(*============================================================================================*)		
(* Collision detection, soll verhinddern, dass nicht gesendet wird, wenn Daten im Empfangsüpuffer sind *)
(* Receive Collision Dectetion *)
bRXCollisionDetected :=	(I_pRxBuffer^.Count > INT_TO_UINT(iMaxBufferBlocking) 
						OR I_pRxBuffer^.FreeByte < (301 -INT_TO_UINT(iMaxBufferBlocking))
						OR I_pRxBuffer^.blocked
						OR I_pRxBuffer^.Error <> 0
						OR fbReceive.StringReceived
						(*OR sReceivedString <> ''*))
						AND bUseRXCollisionDetection;
						
(* Transmit Collision Detection *)
bTXCollisionDetected :=	(I_pTxBuffer^.Count > INT_TO_UINT(iMaxBufferBlocking) 
						OR I_pTxBuffer^.FreeByte < (301 -INT_TO_UINT(iMaxBufferBlocking))
						OR I_pTxBuffer^.blocked
						OR I_pTxBuffer^.Error <> 0)
						AND bUseTXCollisionDetection;
						
(* Collision Detection Verzögern *)						
tonCollisionFree(
	IN := 	NOT bRXCollisionDetected
			AND NOT bTXCollisionDetected,
	PT := 	tVerzCollisionDetect,
	Q =>	bCollisionFree);

(*============================================================================================*)	
(* Ping Intervall Timer *)		
tonPingIntervall(
	IN := I_bAutoPing
			AND NOT bPingStart,
	PT := I_tAutoPingTime);

tonPingVerz(
	PT := I_tVerzPing);	
	
(*============================================================================================*)	
(* Busbelastungstest *)	
bBusBelastungstest := I_bBusBelastungstest;
sReceivedMEMString:='';

(*============================================================================================*)	
(* Anzahl der gefüllten FiFo Zeilen *)
icntFiFo := 0;
iCntFiFoDone := 0;

FOR i := 1 TO cMaxRowCMDFiFo BY 1 DO 
	
	IF i <= I_nMaxDevices
	THEN
		IF (I_sSendCmdFiFo[i]<> '')
		THEN
			icntFiFo := icntFiFo +1;
		END_IF
	END_IF
	
	(* Zählen wie viele Dones gesetzt sind
		wenn alle True sind, ist komplett fertig gesendet *)
	IF i <= I_nMaxDevices
	THEN
		IF Q_bSendDoneFiFo[i]
		THEN
			iCntFiFoDone := iCntFiFoDone +1;
		END_IF
	END_IF
END_FOR

(* Alle FiFo Rows Done *)
bFiFoDone := iCntFiFoDone = I_nMaxDevices;
tonFiFoDoneTimeout.IN :=	NOT bFiFoDone
							AND iStepFiFo = 0;

(*============================================================================================*)	
(* Manuelles Senden *)
rTrigSendManuell(
	CLK := I_bSendManuell);

(*============================================================================================*)
CASE iStepFiFo OF
-1:	sStep := 'FiFo INIT';
	bFirstCycle := FALSE;
	Q_bBusy := FALSE;
	bPingStart := FALSE;
	iFiFoRow := 1;
	iPingRow := 1;
	
	FOR h := 1 TO cMaxRowCMDFiFo BY 1 DO
		IF h <= I_nMaxDevices
		THEN
			Q_bSendDoneFiFo[h] :=TRUE;
		END_IF
	END_FOR
	
	iStepFiFo := 0;

(*============================================================================================*)
0:	sStep := 'Warten, dass FiFo gefüllt wird';
		
	iFiFoRow := 1;
	
	IF iPingRow <= 0
	THEN
		iPingRow := 1;
	END_IF
	
	bStringSend := FALSE;
	Q_bBusy := FALSE;
	tonPingVerz.IN := FALSE;
		
	(* Wenn die Intervall Zeit abgelaufen ist Ping Start setzen *)
	IF tonPingIntervall.Q
	THEN
		bPingStart := TRUE;
	END_IF
	
	(* Notfallschaltung, falls mal ein bDone hängt
		zb. durch Gerätebaustein fehler *)
	IF tonFiFoDoneTimeout.Q
	THEN
		dwCntTimeout := dwCntTimeout+1;
		FOR h := 1 TO I_nMaxDevices BY 1 DO
			Q_bSendDoneFiFo[h] :=TRUE;
		END_FOR
	END_IF
					
	IF bFirstCycle
	THEN
		iStepFiFo := -1;
	ELSE
		IF bCollisionFree
		THEN
			IF icntFiFo > 0
				OR  bBusBelastungstest
				OR I_bManuellMode
			THEN
				(* Normaler Sendevorgang TX *)
				Q_bBusy := TRUE;
				iStepFiFo := 1;
			ELSE
				IF bPingStart
					OR iPingRow < I_nMaxDevices	(* Ping wurde unterbrochen *)
				THEN
					IF iPingRow < I_nMaxDevices
					THEN
						(* Fifo Zeile wieder auf die gespeicherte Ping zeile setzen, weil unterbrochen wurde *)
						iFiFoRow := iPingRow; 
					ELSE
						(* fifo Zeile 1 setzen, weil ende erreicht *)
						iFiFoRow := 1; 
					END_IF
					
					(* Globalen Merker Setzen, dass Ping aktiv ist *)
					bGlobalPingActive := TRUE;
					
					(* Ping senden TX*)
					iStepFiFo := 10;	
				END_IF
			END_IF
		END_IF
	END_IF
	
(*============================================================================================*)	
1:	sStep := 'Prüfen ob STRING in FiFo Zeile gefüllt*';
	
	IF I_bSearchMode
	THEN
		sStep :=fbRS485Search.Q_sState;
	END_IF
	
	(* Manueller Modus *)
	IF I_bManuellMode
	THEN
		(* Prüfen ob in der Zeile etwas steht *)
		IF I_sSendCmdManuell <>''
			AND rTrigSendManuell.Q
			AND NOT I_bSearchMode
		THEN
			IF bCollisionFree
			THEN
				(* Normaler Sendevorgang TX *)
				sString :=	I_sSendCmdManuell; 
				bStringSend := TRUE;
				Q_bDone := FALSE;
				Q_bError := FALSE;
				iStepFiFo := iStepFiFo+1;
			END_IF
		END_IF
		(* Prüfen ob in der Zeile etwas steht *)
		IF I_bSearchMode
			AND fbRS485Search.Q_bSend
		THEN
			IF bCollisionFree
			THEN
				(* Suchmode Sendevorgang TX *)
				sString :=	fbRS485Search.Q_sSearchString; 
				bStringSend := TRUE;
				Q_bDone := FALSE;
				Q_bError := FALSE;
				iStepFiFo := iStepFiFo+1;
			END_IF
		END_IF
	ELSE
		(* Prüfen ob in der ausgewählten Zeile etwas steht *)
		sStringSend :=	I_sSendCmdFiFo[iFiFoRow]; 
		IF I_sSendCmdFiFo[iFiFoRow] = ''
		THEN
			IF iFiFoRow< I_nMaxDevices
			THEN
				iFiFoRow := iFiFoRow+1; (* Nächste Zeile, bis etwas drin Steht *)
			ELSE
				IF bBusBelastungstest
				THEN
					sStringSend :=	CONCAT(F_ToCHR(I_sStartZeichen),'ServiceTOOL-BUSBELASTUNGSTEST-BURSTFIREMODE');
					sStringSend :=	CONCAT(sStringSend,F_ToCHR(I_sEndZeichen));
					(* Senden *)
					
					IF  bCollisionFree
					THEN
						(* Busbelastungstest Sendevorgang TX *)
						sStep := 'Prüfe ob Senden noch aktiv ist';
						bStringSend := TRUE;
						sString :=	sStringSend;
						Q_bDone := FALSE;
						Q_bError := FALSE;
						iStepFiFo := iStepFiFo+1;
					END_IF
				ELSE
					(* Alle Zeilen Abgearbeitet *)
					iStepFiFo := 0;	
				END_IF
			END_IF
		ELSE
		(* Senden *)
		Q_bSendDoneFiFo[iFiFoRow] :=FALSE;
		
			IF bCollisionFree
			THEN
				(* Normaler Sendevorgang TX *)
				sStep := 'Prüfe ob Senden noch aktiv ist';
				bStringSend := TRUE;
				sString :=	sStringSend;
				Q_bDone := FALSE;
				Q_bError := FALSE;
				iStepFiFo := iStepFiFo+1;
			END_IF
		END_IF
	END_IF
	
(*============================================================================================*)		
2:	sStep := 'Starte Senden';
	Q_bBusy := TRUE;
	tonTimeout.IN := fbSend.Busy;
	
	IF NOT fbSend.Busy
		AND NOT fbReceive.StringReceived
	THEN	
		(* Normaler Sendevorgang TX *)
		sString := '';
		tonSend.IN := FALSE;
		bStringSend := FALSE;
		iStepFiFo := iStepFiFo+1;
	ELSIF
		(fbSend.Error >0)
		AND NOT (fbSend.Error = 2)
	THEN
		sStep := CONCAT('ERROR-',sStep);
		sStep := CONCAT(sStep,'- ');
		sStep := CONCAT(sStep,INT_TO_STRING(fbSend.Error));
		iStepFiFo := -2;
	ELSIF
		tonTimeout.Q
	THEN
		sStep := CONCAT('ERROR- Timeout',sStep);
		iStepFiFo := -2;
	END_IF
	
(*============================================================================================*)		
3:	(* Senden*)		
	Q_bSendDoneFiFo[iFiFoRow] :=TRUE;
	
	IF iFiFoRow< I_nMaxDevices
		AND NOT I_bSearchMode
	THEN
		iFiFoRow := iFiFoRow+1;
		iStepFiFo := 1;
	ELSE
		Q_bDone := TRUE;
		
		IF (NOT fbRS485Search.Q_bSend
			AND I_bSearchMode)
			OR NOT I_bSearchMode
		THEN
			iStepFiFo := 0;
		END_IF
	END_IF
	
(*============================================================================================*)	
(* Ping Senden Ablauf *)
(*============================================================================================*)	
10:	sStep := 'Sende Ping*';
	
	tonPingVerz.IN := FALSE;
	
	(* Ping String erstellen *)
	sStringSend:=	CONCAT(F_ToCHR(I_sStartZeichen),DINT_TO_STRING(I_stDeviceIdent[iFiFoRow].diID));
	sStringSend :=	CONCAT(sStringSend,'.');
	sStringSend :=	CONCAT(sStringSend ,I_stDeviceIdent[iFiFoRow].sPingIdent); 
	sStringSend :=	CONCAT(sStringSend,F_ToCHR(I_sEndZeichen));
	
	IF I_stDeviceIdent[iFiFoRow].sPingIdent = ''
		OR I_stDeviceIdent[iFiFoRow].diID = 0
	THEN
		IF iFiFoRow < I_nMaxDevices
		THEN
			iFiFoRow := iFiFoRow+1; (* Nächste Zeile, bis etwas drin Steht *)
		ELSE
			bPingStart := FALSE;
			iPingRow := I_nMaxDevices;
			iStepFiFo := 0;	(* Alle Zeilen Abgearbeitet *)
		END_IF
	ELSE
	(* Senden *)	
		IF bCollisionFree
		THEN
			sStep := 'Prüfe ob Senden noch aktiv ist';
			bStringSend := TRUE;
			sString :=	sStringSend;
			Q_bDone := FALSE;
			Q_bError := FALSE;
			iStepFiFo := iStepFiFo+1;
		END_IF
	END_IF
	
(*============================================================================================*)		
11:	sStep := 'Starte Senden';
	Q_bBusy := TRUE;
	tonTimeout.IN := fbSend.Busy;
	
	IF NOT fbSend.Busy
		(*AND NOT fbReceive.StringReceived*)
	THEN
		tonSend.IN := FALSE;
		bStringSend := FALSE;
				
		IF NOT fbReceive.StringReceived
			AND bCollisionFree
		THEN
			iStepFiFo := iStepFiFo+1;
		END_IF
		
	ELSIF
		(fbSend.Error >0)
		AND NOT (fbSend.Error = 2)
	THEN
		sStep := CONCAT('ERROR-',sStep);
		sStep := CONCAT(sStep,'- ');
		sStep := CONCAT(sStep,INT_TO_STRING(fbSend.Error));
		iStepFiFo := -2;
	ELSIF
		tonTimeout.Q
	THEN
		sStep := CONCAT('ERROR- Timeout',sStep);
		iStepFiFo := -2;
	END_IF
	
(*============================================================================================*)		
12:	(* Senden*)		
	(* Nur speichern wenn auch wirklich eine ID vorhanden ist *)	
	IF I_stDeviceIdent[iFiFoRow].sPingIdent = ''
		OR I_stDeviceIdent[iFiFoRow].diID = 0
	THEN
		IF iFiFoRow < I_nMaxDevices
		THEN
			iFiFoRow := iFiFoRow+1; (* Nächste Zeile, bis etwas drin Steht *)
		ELSE
			bGlobalPingActive := FALSE;
			bPingStart := FALSE;
			iPingRow := I_nMaxDevices;
			iStepFiFo := 0;	(* Alle Zeilen Abgearbeitet *)
		END_IF
	ELSE
		IF iFiFoRow < I_nMaxDevices
		THEN
			iFiFoRow := iFiFoRow+1;
			iPingRow := iFiFoRow; (* Zeile speichern *)
			iStepFiFo := 13;	(* Falls das warten Deaktiviert werden soll, kann hier einfach in 10 gesprungen werden *)
		ELSE
			bPingStart := FALSE; (* Letzte Ping Zeile erreicht, Timer zurücksetzen  *)
			iPingRow := I_nMaxDevices;
			iStepFiFo := 13;
		END_IF
	END_IF
(*============================================================================================*)		
13:	(* Optionale Wartezeit zwischen jedem Ping*)		
	tonPingVerz.IN := TRUE;
			
	IF tonPingVerz.Q
	THEN
		IF NOT fbReceive.StringReceived
			AND bCollisionFree
		THEN
			tonPingVerz.IN := FALSE;
			
			IF iFiFoRow < I_nMaxDevices
			THEN
				iStepFiFo := 10; (* nächsten Ping senden *)
			ELSE
				bGlobalPingActive := FALSE;
				iStepFiFo := 0;
			END_IF
		END_IF
	ELSE
		(* Prüfen ob ein Sendeauftrag anliegt *)
		IF icntFiFo >0
		THEN
			tonPingVerz.IN := FALSE;
			iStepFiFo := 0; (* Sende FiFo leeren *)
		END_IF  
	END_IF
ELSE
(*============================================================================================*)
	Q_bError := TRUE;
	Q_bBusy := FALSE;
	bBusyMem := FALSE;
	tonTimeout.IN := FALSE;
	
	IF I_bReset
	THEN
		iStepFiFo := 0;
	END_IF
END_CASE

(*============================================================================================*)	
(* Nur Senden, wenn nicht Empfangen wird *)
IF bStringSend
THEN
	IF bActivateSend
	THEN
		(* Senden *)
		fbSend(
			SendString:= 	sString,
			TXbuffer:= 		I_pTxBuffer^);
	END_IF
	
ELSE
	IF bActivateReceive
	THEN
		(* Empfangen *)
		ac00_Receive();
	END_IF
END_IF

(*============================================================================================*)	
(* Empfangsmerker 0 Setzen am ende Eines Zyklus *)
Q_sReceiveString := sReceivedMEMString;

(*============================================================================================*)	
(* Busauslastung tracken*)
ac99_Diagnose();

(*============================================================================================*)	
(* StatusStruktur für Visu *)
Q_sState :=	sStep;
Q_stStates.bBusy				:=	Q_bBusy;
Q_stStates.bDone				:=	Q_bDone;
Q_stStates.bError				:=	Q_bError;
Q_stStates.iFiFoCount			:=	icntFiFo;
Q_stStates.iFiFoRow				:=	iFiFoRow;
Q_stStates.lrBusAuslastung		:=	Q_lrBusAuslastung;
Q_stStates.sReceiveString 		:=	Q_sReceiveString;
Q_stStates.sSendString 			:=	sString;
Q_stStates.sState 				:=	Q_sState;

(*============================================================================================*)	
(* RS485 Telegramm Logging *)
fbRS485Logger(
	I_bExecute:= 		I_bLogger,						(* oder eine externe Variable *)
	I_bReset:=			I_bResetLog,	
	I_sTxTelegram:= 	sString,
	I_sRxTelegram:= 	sReceivedMEMString);

ACTION ac00_Receive:
(*============================================================================================*)	
(* Empfangen *)

CASE iStepReceive OF		
0:	fbReceive(
		Prefix := 			F_ToCHR(I_sStartZeichen),
		Suffix := 			F_ToCHR(I_sEndZeichen),
		Timeout:= , 
		Reset:= , 
		StringReceived=> , 
		Busy=> , 
		Error=> , 
		RxTimeout=> , 
		ReceivedString:= 	sReceivedString, 
		RXbuffer:= 			I_pRxBuffer^);
		
	IF fbReceive.StringReceived
	THEN
		iStepReceive := 1;
		sReceivedMEMString := sReceivedString;
	END_IF
	
1:	sReceivedString := '';
	iStepReceive := 0;

	
END_CASE
END_ACTION

ACTION ac99_Diagnose:
(*============================================================================================*)	
(* Busauslastung Prüfen *)

fbBusAuslastung(
	I_bExcecute:= 	bBusAuslastung, 
	I_nWert:= 		UINT_TO_LREAL(I_pTxBuffer^.Count), 
	I_nFilterWert:= 50, 
	Q_nFilter=> 	Q_lrBusAuslastung);
	
	
fbRS485Search(
	I_bStartSearch:= 	I_bSearchMode, 
	I_diStartID:= , 
	I_diMaxID:= , 
	I_sStartZeichen:= 	I_sStartZeichen, 
	I_sEndZeichen:= 	I_sEndZeichen, 
	I_tWait:= , 
	I_StringReceived:= 	sReceivedMEMString, 
	Q_bSend=> , 
	Q_sSearchString=> );
END_ACTION

END_FUNCTION_BLOCK

// ---- POUs/RS485_Hausbus_FB/00_RS485 COM/RS485_Master/fb_RS485Logger.TcPOU
(*======================================================================================================================================*)
(*//=============================================================================\\
||  _   _ _  __  _         _                        _   _                      ||
|| | \ | | |/ / / \  _   _| |_ ___  _ __ ___   __ _| |_(_) ___  _ __         ||
|| |  \| | ' / / _ \| | | | __/ _ \| '_ ` _ \ / _` | __| |/ _ \| '_ \        ||
|| | |\  | .  \/ ___ \ |_| | || (_) | | | | | | (_| | |_| | (_) | | | |       ||
|| |_| \_|_|\_\_/  \_\__,_|\__\___/|_| |_| |_|\__,_|\__|_|\___/|_| |_|       ||
||                                                                             ||
\\=============================================================================//*)
(*fb_RS485Logger: 	Einfaches Logging von RX und TX Telegrammen*)
(*
Date          	| Version    	| created under        	| Author          	| Remark *)
(*====================================================================================================================================================*)
(*11/01/2026   	| 1.00      		| TC3		  		| N. Kersting       | first release *)
(*11/01/2026   	| 1.01      		| TC3		  		| N.  Kersting       | Ringbuffer implementiert - neueste oben *)
(*11/01/2026   	| 1.02      		| TC3		  		| N.  Kersting       | Array wird geleert wenn Execute FALSE ist *)
(*12/01/2026   	| 1.03      		| TC3		  		| N.  Kersting       | Reset eingang zum zurücksetzen des gesamten Arrays *)
(*====================================================================================================================================================*)
FUNCTION_BLOCK fb_RS485Logger
VAR_INPUT
	I_bExecute				: BOOL := TRUE;								(* Enable/Disable Logging *)
	I_bReset				: BOOL;										(* Reset Log Buffer *)
	I_sTxTelegram			:STRING(255);								(* TX Telegramm zum Logging *)
	I_sRxTelegram			:STRING(255);								(* RX Telegramm zum Logging *)
END_VAR
VAR_OUTPUT
	Q_asLogBuffer			:ARRAY[1..50] OF STRING(255);				(* Log Buffer mit max.  200 Zeilen *)
	Q_iLogIndex				:INT;										(* Aktuelle Index Position *)
	Q_iLogCount				:INT;										(* Anzahl der geloggten Einträge *)
END_VAR
VAR
	sTxLast					: STRING(255) := '';						(* Letzter TX String zum Vergleich *)
	sRxLast					: STRING(255) := '';						(* Letzter RX String zum Vergleich *)
	bExecuteLast			: BOOL := TRUE;								(* Letzter Execute Status *)
	iWriteIndex				: INT := 1;									(* Schreibposition Ringbuffer *)
	iLogCount				:INT := 0;									(* Gesamtanzahl Logs *)
	sLogEntry				: STRING(255);								(* Temporärer Log Eintrag *)
	i, h					: INT;										(* Zähler *)

END_VAR

(*============================================================================================*)
(* Reset Log Buffer - leert das komplette Array *)
IF I_bReset
THEN
	FOR i := 1 TO 50 BY 1 DO
		Q_asLogBuffer[i] := '';
	END_FOR
	iLogCount := 0;
	sTxLast := '';
	sRxLast := '';
	RETURN;
END_IF

(*============================================================================================*)
(* Logging deaktiviert - nur schreiben pausieren *)
IF NOT I_bExecute
THEN
	RETURN;
END_IF

(*============================================================================================*)
(* TX Telegramm Logging *)
IF I_sTxTelegram <> '' 
	AND I_sTxTelegram <> sTxLast
THEN
	(* Alle Zeilen nach unten verschieben - rückwärts von 199 bis 1 *)
	FOR h := 49 TO 1 BY -1 DO
		Q_asLogBuffer[h + 1] := Q_asLogBuffer[h];
	END_FOR
	
	(* Neuer Eintrag oben *)
	sLogEntry := CONCAT('TX: ', I_sTxTelegram);
	Q_asLogBuffer[1] := sLogEntry;
	sTxLast := I_sTxTelegram;
	
	(* Counter erhöhen, aber max. 200 *)
	IF iLogCount < 50
	THEN
		iLogCount := iLogCount + 1;
	END_IF
END_IF

(*============================================================================================*)
(* RX Telegramm Logging *)
IF I_sRxTelegram <> '' 
	AND I_sRxTelegram <> sRxLast
THEN
	(* Alle Zeilen nach unten verschieben - rückwärts von 199 bis 1 *)
	FOR h := 49 TO 1 BY -1 DO
		Q_asLogBuffer[h + 1] := Q_asLogBuffer[h];
	END_FOR
	
	(* Neuer Eintrag oben *)
	sLogEntry := CONCAT('RX: ', I_sRxTelegram);
	Q_asLogBuffer[1] := sLogEntry;
	sRxLast := I_sRxTelegram;
	
	(* Counter erhöhen, aber max. 200 *)
	IF iLogCount < 50
	THEN
		iLogCount := iLogCount + 1;
	END_IF
END_IF

(*============================================================================================*)
(* Output Parameter aktualisieren *)
Q_iLogCount := iLogCount;

END_FUNCTION_BLOCK

// ---- POUs/RS485_Hausbus_FB/00_RS485 COM/RS485_Master/fb_RS485Startup.TcPOU
(*======================================================================================================================================*)
(*//=============================================================================\\
||  _   _ _  __  _         _                        _   _                      ||
|| | \ | | |/ / / \  _   _| |_ ___  _ __ ___   __ _| |_(_) ___  _ __         ||
|| |  \| | ' / / _ \| | | | __/ _ \| '_ ` _ \ / _` | __| |/ _ \| '_ \        ||
|| | |\  | . \/ ___ \ |_| | || (_) | | | | | | (_| | |_| | (_) | | | |       ||
|| |_| \_|_|\_\_/  \_\__,_|\__\___/|_| |_| |_|\__,_|\__|_|\___/|_| |_|       ||
||                                                                             ||
\\=============================================================================//
fb_RS485Startup:	Einfacher Baustein um die Hardware für die RS485 Haus-Bus vorzubereiten*)
(*
Date          	| Version    	| created under        	| Author          	| Remark *)
(*====================================================================================================================================================*)
(*13/05/2025   	| 1.00      		| TC3		  		| N.Kersting       | first release *)
(*18/08/2025   	| 1.01      		| TC3		  		| N.Kersting       | Startup über bExecute nun erneut Anwählbar*)
(*13/10/2025   	| 1.02      		| TC3		  		| N.Kersting       | Automatische Quittierung bei Busfehler*)
(*15/10/2025   	| 1.03      		| TC3		  		| N.Kersting       | Spannungsversorgung nun steuerbar über diesen Baustein*)
(*19/10/2025   	| 1.04      		| TC3		  		| N.Kersting       | Bugfix automatische Quittierung nach Busfehler nur bei Spannung Ok*)
(*====================================================================================================================================================*)
FUNCTION_BLOCK fb_RS485Startup
VAR_INPUT
	I_bExecute						:BOOL;
	I_bBusOK						:BOOL;
	I_bSpannungOk					:BOOL;
	I_bStandby						:BOOL;
	I_tStartupVerz					:TIME := T#2S;	(* Startup verzögert ausführen *)
END_VAR
VAR_IN_OUT
	IQ_InData	 					:KL6inData22B;
    IQ_OutData						:KL6outData22B;
END_VAR
VAR_OUTPUT
	Q_sState						:STRING;
	Q_bStartupDone					:BOOL;
	Q_bError						:BOOL;
	Q_bSpannungEin					:BOOL;
	Q_bSpannungAus					:BOOL;
	Q_stStates						:ST_RS485Startup_State;
END_VAR
VAR
	udBaudrate						:UDINT := 57600;
	byDataBits						:BYTE := 8;
	byStopBits						:BYTE := 1;
	
	tonStartupVerz					:ton;
	tonTimeout						:ton;
	fbSerialComReset				:ComReset;
	fComBufferReset					:ClearComBuffer;
	fbSerialConfig 					:KL6Configuration;  // Terminal-Konfiguration (Baud, Parität etc.)
	iStepStartup					:INT;
	rTrigStartupStart				:r_trig;
	bBusFehlerMerker				:BOOL;
END_VAR

tonStartupVerz(
	PT :=	I_tStartupVerz);

tonTimeout();	

rTrigStartupStart(CLK :=Q_bStartupDone
						AND I_bExecute
						AND I_bBusOK);
	
CASE iStepStartup OF 
(*=========================================================================*)
0:	tonTimeout.IN := FALSE;
	Q_bSpannungEin := FALSE;
	Q_bSpannungAus := FALSE;
	
	IF NOT Q_bError
		AND I_bBusOK
	THEN
		Q_sState := 'INIT';
	ELSIF
		NOT I_bBusOK
	THEN
		bBusFehlerMerker := TRUE;
		Q_bError := TRUE;
		Q_sState := 'Busverbindung nicht Ok';
	END_IF
	
	tonStartupVerz.IN := FALSE;
	
	fbSerialComReset(
		Execute:= 		FALSE);
		
	fbSerialConfig(
		Execute:= 		FALSE);
		
	(* Automatische Quittierung nach Busfehler *)
	IF bBusFehlerMerker
		AND I_bBusOK
		AND I_bSpannungOk
	THEN
		Q_bStartupDone := FALSE;
		iStepStartup := iStepStartup+1;
	END_IF
	
	IF I_bExecute
		AND I_bBusOK
		AND I_bSpannungOk
	THEN
		Q_bStartupDone := FALSE;
		iStepStartup := iStepStartup+1;
	ELSIF
		I_bExecute
		AND I_bBusOK
		AND NOT I_bSpannungOk
	THEN
		Q_bStartupDone := FALSE;
		iStepStartup := 100;
	END_IF

(*=========================================================================*)
1:	Q_sState := 'Warten auf Verzögerung';
	tonStartupVerz.IN := TRUE; 
	
	IF tonStartupVerz.Q
	THEN
		iStepStartup := iStepStartup+1;
	END_IF
	
(*=========================================================================*)
2:	Q_sState := 'Serielle Klemme Konfigurieren mit Haus-Bus Vorgaben';	
	
	fbSerialConfig(
		Execute:= 		TRUE, 
		Mode:= 			ComSerialLineMode_t.SERIALLINEMODE_KL6_22B_STANDARD,		 
		Baudrate:= 		udBaudrate, 
		NoDatabits:= 	byDataBits, 
		Parity:= 		ComParity_t.PARITY_EVEN,	 
		Stopbits:= 		byStopBits, 
		Handshake:= 	RS485_HALFDUPLEX, 
		ContinousMode:= , 
		pComIn := 		ADR(IQ_InData), 
		pComOut := 		ADR(IQ_OutData), 
		SizeComIn := 	SIZEOF(IQ_InData),
		Done=> , 
		Busy=> , 
		Error=> , 
		ErrorId=> );
	
	IF fbSerialConfig.Done
	THEN
		fbSerialConfig(
			Execute:= 		FALSE); 
			
		iStepStartup := 3;
	ELSIF
		fbSerialConfig.Error
	THEN
		Q_sState := 'Error fbSerialConfig ID: ';
		Q_sState := CONCAT(Q_sState,INT_TO_STRING(fbSerialConfig.ErrorID));
		iStepStartup := -2;	//Error
	END_IF

(*=========================================================================*)
3:	Q_sState := 'Serielle Klemme Reset Auführen';	
		
	fbSerialComReset(
		Execute:= 		TRUE, 
		pComIn := 		ADR(IQ_InData), 
		pComOut := 		ADR(IQ_OutData), 
		SizeComIn := 	SIZEOF(IQ_InData),
		Done=> , 
		Busy=> , 
		Error=> , 
		ErrorID=> );	
		
	IF fbSerialComReset.Done
	THEN
		iStepStartup := 999;
	ELSIF
		fbSerialComReset.Error
	THEN
		Q_sState := 'Error fbSerialComReset ID: ';
		Q_sState := CONCAT(Q_sState,INT_TO_STRING(fbSerialComReset.ErrorID));
		iStepStartup := -3;	//Error
	END_IF

(*=========================================================================*)
100:Q_sState := 'Spannung einschalten';
	tonTimeout.IN := TRUE;
	tonTimeout.PT := T#5S;
	
	Q_bSpannungEin := TRUE;

	IF 	I_bSpannungOk
	THEN
		Q_bSpannungEin := FALSE;
		tonTimeout.IN := FALSE;
		iStepStartup := 1;
	ELSIF
		tonTimeout.Q
	THEN
		Q_bSpannungEin := FALSE;
		tonTimeout.IN := FALSE;
		Q_sState := 'Timeout Spannung einschalten';
		iStepStartup := -100;
	END_IF

(*=========================================================================*)
200:Q_sState := 'Spannung ausschalten';
	tonTimeout.IN := TRUE;
	tonTimeout.PT := T#5S;
	
	Q_bSpannungAus := TRUE;

	IF 	NOT I_bSpannungOk
	THEN
		Q_sState := 'HausBus Spannung über Standby Ausgeschaltet. Startup Ausführen zum einschalten!';
		Q_bSpannungAus := FALSE;
		tonTimeout.IN := FALSE;
		iStepStartup := -201;	(* Standby *)
	ELSIF
		tonTimeout.Q
	THEN
		Q_bSpannungAus := FALSE;
		tonTimeout.IN := FALSE;
		Q_sState := 'Timeout Spannung ausschalten';
		iStepStartup := -200;
	END_IF
	
(*=========================================================================*)
999:Q_sState := 'Startup Ausgeführt!';	
	Q_bStartupDone := TRUE;
	Q_bError := FALSE;
	bBusFehlerMerker := FALSE;
	tonTimeout.IN := FALSE;
	Q_bSpannungEin := FALSE;
	Q_bSpannungAus := FALSE;
	
	IF NOT I_bBusOK
		OR NOT I_bSpannungOk
	THEN
		bBusFehlerMerker := TRUE;
		Q_bStartupDone := FALSE;
		iStepStartup := 0;
	END_IF
	
	IF I_bSpannungOk
		AND I_bStandby
	THEN
		Q_bStartupDone := FALSE;
		iStepStartup := 200;
	END_IF
	
	IF rTrigStartupStart.Q
	THEN
		Q_bStartupDone := FALSE;
		iStepStartup := 1;
	END_IF

ELSE
	(* ERROR *)
	Q_bError := TRUE;
	iStepStartup := 0;
END_CASE

(* StatusStruktur für Visu *)
Q_stStates.bBusOk				:=	I_bBusOK;
Q_stStates.bStartupDone			:=	Q_bStartupDone;
Q_stStates.bStartupError		:=	Q_bError;
Q_stStates.sStartupState		:=	Q_sState;

END_FUNCTION_BLOCK

// ---- POUs/RS485_Hausbus_FB/01_BusTaster/fb_TasterBus6F.TcPOU
(*======================================================================================================================================*)
(*//=============================================================================\\
||  _   _ _  __  _         _                        _   _                      ||
|| | \ | | |/ / / \  _   _| |_ ___  _ __ ___   __ _| |_(_) ___  _ __         ||
|| |  \| | ' / / _ \| | | | __/ _ \| '_ ` _ \ / _` | __| |/ _ \| '_ \        ||
|| | |\  | . \/ ___ \ |_| | || (_) | | | | | | (_| | |_| | (_) | | | |       ||
|| |_| \_|_|\_\_/  \_\__,_|\__\___/|_| |_| |_|\__,_|\__|_|\___/|_| |_|       ||
||                                                                             ||
\\=============================================================================//
fb_TasterBus6F:	Einfache RS485 Kommunikation für Haus-bus.de Komponenten zum testen 	
				Achtung: Bei dem 6 Fach Taster ist zu Beachten, dass es nur 4 Externe EA/s gibt also 4 LEDs und 4 Taster *)
(*
Date          	| Version    	| created under        	| Author          	| Remark *)
(*====================================================================================================================================================*)
(*29/04/2025   	| 1.00      		| TC3		  		| N.Kersting       | first release *)
(*02/05/2025   	| 1.01      		| TC3		  		| N.Kersting       | Events für die Buttons werden erfolgreich verarbeitet *)
(*02/05/2025   	| 1.02      		| TC3		  		| N.Kersting       | Events für Temp, Helligkeit, Fuehctigkeit erfolgreich Implementier *)
(*02/05/2025   	| 1.03      		| TC3		  		| N.Kersting       | Set Schrittkette für Reset und LED Helligkeit erfolgreich Implementier*)
(*02/05/2025   	| 1.04      		| TC3		  		| N.Kersting       | In und Out Strukturen Implementiert und Startup nach Reset *)
(*02/05/2025   	| 1.05      		| TC3		  		| N.Kersting       | Pingabgfrage*)
(*02/05/2025   	| 1.06      		| TC3		  		| N.Kersting       | Reset Startup Implementiert*)
(*03/05/2025   	| 1.07      		| TC3		  		| N.Kersting       | Ping wird nun bei PLC Reset auch gestaret und Execute wird richtig verwendet*)
(*04/05/2025   	| 1.08      		| TC3		  		| N.Kersting       | Hintergrundbeleuchtung und Zähler für die Tatser Implementiert *)
(*04/05/2025   	| 1.09      		| TC3		  		| N.Kersting       | Neuen Baustein zum Einheitlichen versenden von Telegrammen Implementiert *)
(*05/05/2025   	| 2.00      		| TC3		  		| N.Kersting       | Komplett neuen Baustein, mit Externer Receive Auswertung und neuem Ping Baustein *)
(*06/05/2025   	| 2.01      		| TC3		  		| N.Kersting       | Externe LEDs Implementiert *)
(*07/05/2025   	| 2.02      		| TC3		  		| N.Kersting       | Im Startup wird nun auf die Device ID geachtet *)
(*08/05/2025   	| 2.03      		| TC3		  		| N.Kersting       | Externe LEDs sind nun Umschaltbar/ LEDs oder normaler Ausgang (Betriefft die Hintergrundbeleuchtung) -> Weniger Busauslastung *)
(*09/05/2025   	| 2.04      		| TC3		  		| N.Kersting       | Ping Versuche Implementiert mit Globalen Parametern *)
(*09/05/2025   	| 2.05      		| TC3		  		| N.Kersting       | Ping für Taster nun Auch automatisch durch Empfang von sämtlichen Telegrammen*)
(*09/05/2025   	| 2.06      		| TC3		  		| N.Kersting       | Bugfix im Startup Angepasst! nur noch Hintergrundbeleuchtung setzen! *)
(*10/05/2025   	| 3.00      		| TC3		  		| N.Kersting       | Umstellung auf Externe FiFo Sendebaustein *)
(*13/05/2025   	| 3.01      		| TC3		  		| N.Kersting       | Viele Bugs gefixt, bei Änderung der Ausgängen wird nun eine Anforderung gesetzt  *)
(*13/05/2025   	| 3.02      		| TC3		  		| N.Kersting       | Test für Github *)
(*23/05/2025   	| 3.03      		| TC3		  		| N.Kersting       | Auto - Input Fault Detection implementiert (Wenn Taster zu lange aktiviert bleibt ) *)
(*28/05/2025   	| 3.04      		| TC3		  		| N.Kersting       | Neuen Einfachen Ping Baustein, welcher nicht sendet, nur auswertet implementiert *)
(*14/08/2025   	| 3.05      		| TC3		  		| N.Kersting       | Neuen Taster Eventbaustein, welcher deutlich weniger CPU Last verursacht  *)
(*27/08/2025   	| 4.00      		| TC3		  		| N.Kersting       | Neue Startupschrittkette sollte alle Eventbausteine auch Resetten  *)
(*28/08/2025   	| 5.00      		| TC3		  		| N.Kersting       | Komplett neue Evolutionsstufe, alle Hausbusgeräte werden nun vom fb_UniHBComOperator gesteuert  *)
(*28/08/2025   	| 5.01      		| TC3		  		| N.Kersting       | Etrster Test erfogreich *)
(*31/08/2025   	| 5.02      		| TC3		  		| N.Kersting       | Bugfix OP Mode wird angezeigt bei Init *)
(*03/09/2025   	| 5.03      		| TC3		  		| N.Kersting       | Events geben nun einen Zeitstempel und die differenz vom letzten Update aus *)
(*05/09/2025   	| 5.04      		| TC3		  		| N.Kersting       | Changecounter gibt nun die Anzahl der  Startups wieder *)
(*09/09/2025   	| 5.05      		| TC3		  		| N.Kersting       | Events aus der For-schleife geholt *)
(*29/09/2025   	| 5.06      		| TC3		  		| N.Kersting       | Inputfault detection für Ext eingänge deaktiviert für Bewegungsmelder *)
(*22/01/2026   	| 7.00      		| TC3		  		| N.Kersting       | Komplett überarbeitet mit umstellung auf Stringbuilder *)
(*25/01/2026   	| 7.01      		| TC3		  		| N.Kersting       | Eventbausteine alle komplett überarbeitet mit den neuen ASCII_RS485 Funktionen *)
(*08/06/2026   	| 8.00      		| TC3		  		| N.Kersting       | Vorbereitung für Bibliotheksfähigkeit, keine externen Referenzen mehr *)
(*20/09/2026   	| 9.00      		| TC3		  		| N.Kersting       | Selbsttest für Abfrage der eingänge *)
(*20/09/2026   	| 9.01      		| TC3		  		| N.Kersting       | Selbsttest Bugfix Schrittkette *)
(*20/09/2026   	| 9.02      		| TC3		  		| N.Kersting       | Selbsttest Bugfix Schrittkette *)
(*20/09/2026   	| 9.03      		| TC3		  		| N.Kersting       | Selfcheck nun nur, wenn Globaler Pingmerker nicht aktiv *)
(*20/09/2026   	| 9.04      		| TC3		  		| N.Kersting       | Kleine anpassung Autoping *)
(*====================================================================================================================================================*)
FUNCTION_BLOCK fb_TasterBus6F
VAR_INPUT
	I_bUsePing			:BOOL;
	I_tPingTime			:TIME := T#15S;
	I_tSelfCheckTime	:TIME := T#15S;
	
	I_bFiFoDone			:BOOL;
	I_FifoID			:INT;
	I_bPingStart		:BOOL;						(* Ping Done vom Vorheriegen*)
	I_bSelfCheck		:BOOL := FALSE;				(* 1x Eingänge prüfen Achtung Flanke!*)
	I_bSelfCheckAuto	:BOOL := FALSE;				(* Eingänge Automatisch Intervallsmäßig prüfen *)
	
	I_stInput			:ST_BusTaster6F_Input;
	I_StringReceived	:STRING(255);
END_VAR
VAR_OUTPUT
	Q_sFiFoSend			:STRING(255);
   	Q_stOutput			:ST_BusTaster6F_Output;
	Q_stCnt				:ST_BusTaster6F_Cnt;
END_VAR
VAR
(*----------------------------------------------*)
(* Interne Parameter*)
(*----------------------------------------------*)		
	bSetExecute			:BOOL := TRUE;				(* Aktiviert die Schrittketten, welche Telegramme versenden *)
	bCheckPing			:BOOL := TRUE;				(* Ping Checken Schrittkette Aktivieren *)
	bInputFaultDetect	:BOOL := TRUE;				(* Prüft die Eingänge ob sie zu lange geschaltet wurden und führt ein reset des eingangs aus *)
	
	sStartZeichen		:BYTE := 16#FD;				(* Startzeichen Präfix *)
	sEndZeichen			:BYTE := 16#FE;				(* Endzeichen Suffix *)
	
	tPingTimer			:TIME:= T#5S;				(* Zeit, bis wiederholend der Ping versendet wird *)
	tStartupLEDOn		:TIME:= T#4S;				(* Zeit, wie Lange die LEDS beim Startup kurz eingeschaltet werden *)
	tResetTimeout		:TIME:= T#10S;				(* Zeit, bis bei einem Reset es zu einem Fehler kommt, wenn kein Ping empfangen wird *)
	tResetReboot		:TIME:= T#10S;				(* Zeit, die nach einem Reset Abgewaretet wird damit das Gerät neustarten kann*)
	tStartupAfterReset	:TIME := T#5S;				(* Zeit, wann das Startup Zurückgesetzt wird, wenn der Ping verloren wird *)
	tInputFaultDetect	:TIME := T#10S;				(* Prüft die Eingänge ob sie zu lange geschaltet wurden und führt ein reset des eingangs aus *)
	
	tSelfCheckStatus	:TIME := T#15S;				(* Prüft die Externen u. Internen Eingänge zyklisch in diesem rythmus ab *)
(*----------------------------------------------*)
(* Strings *)
(*----------------------------------------------*)			
	sSendString			:STRING(255);
	sFiFoSend			:STRING(255);
	sReceived			:STRING(255);
	sLastSendString		:STRING(255);
	sStateReset			:STRING;
(*----------------------------------------------*)
(* Funktionsbausteine *)
(*----------------------------------------------*)
	fbUniHBComOperator	:fb_UniHBComOperator;
	fbBusTasterEventExt	:fb_BusTasterAdvancedEvent_6F;
	fbBusTasterEvent	:fb_BusTasterAdvancedEvent_6F;
	fbBusTempEvent		:fb_BusTempEvent;
	fbBusBrsEvent		:fb_BusBrsEvent;
	fbBusRhdEvent		:fb_BusRhdEvent;
	fbBusPingEvent		:fb_BusPingEvent;
(*----------------------------------------------*)
(* Indexe *)
(*----------------------------------------------*)	
	iStepSet			:INT;
	i,h,j,l,e			:INT;
	
	iDimmMem			:ARRAY[1..6] OF INT;
	iDimmMemExt			:ARRAY[1..6] OF INT;
	iDimmBGAnf			:INT;
	iDimmAnf			:ARRAY[1..6] OF INT;
	iDimmAnfExt			:ARRAY[1..6] OF INT;
	
	iDimmBgMem			:INT;
	cntChangesDimm		:INT;
	cntChangesDimmExt	:INT;
(*----------------------------------------------*)
(* Timer/Trigger *)
(*----------------------------------------------*)		
	r_TrigReset				:r_trig;		
	r_TrigCountBtn			:ARRAY[1..6] OF r_trig;
	
	tonResetTimeout			:ton;
	tonStepStartup			:ton;
	tonSelfCheck			:ton;
(*----------------------------------------------*)
(* Status *)
(*----------------------------------------------*)			
	bMemExt					:BOOL;
	bSendeAnforderung		:BOOL;
	bSendeAnforderungExt	:BOOL;
	bSendeAnforderungBG		:BOOL;
	bErrorReset				:BOOL;
	bResetBusy				:BOOL;
	bResetDone				:BOOL;
	bStartupDone			:BOOL;
	bEventStartupDone		:BOOL;
	bSelfCheckAnforderung	:BOOL;
	
	fbRS485HBStringBuilder	:fb_RS485HB_StringBuilder;
END_VAR

(*///////////////////////////////////////////////////////////*)
(* Parameter *)
tPingTimer :=			I_tPingTime;
bCheckPing :=			I_bUsePing;

(*///////////////////////////////////////////////////////////*)
(* Reset *)
r_TrigReset(CLK := 	I_stInput.bReset);

(*///////////////////////////////////////////////////////////*)
(* Ident beschreiben *)
fbUniHBComOperator.I_stIdent.bUseExtInputs 	:=	I_stInput.bExtInputs;
fbUniHBComOperator.I_stIdent.diID 			:=	I_stInput.diID;
fbUniHBComOperator.I_stIdent.sName 			:=	I_stInput.sName;

(*///////////////////////////////////////////////////////////*)
(*	Operator *)
fbUniHBComOperator(
	I_bExtInputs:= 			I_stInput.bExtInputs, 
	I_bExecute:= 			I_stInput.bExecute
							AND NOT r_TrigReset.Q, 
	I_bPing:= 				fbBusPingEvent.Q_bOut, 
	I_bPingCheck:=			I_bPingStart,
	I_bEventStartupDone:= 	bEventStartupDone, 
	I_bResetSendDone:= 		bResetDone,	 
	I_bStartupDone:= 		bStartupDone, 
	I_tPingTimeout:= 		tPingTimer, 
	I_tStartupAfterReset:= 	tStartupAfterReset, 
	I_tReboot:=				tResetReboot,
	Q_EState=> 				,			 
	Q_bResetEvents=> 		, 
	Q_bExecuteEvents=> 		, 
	Q_bSendResetCmd=> 		, 
	Q_bStartupStart=> 		, 
	Q_bActivateSend=>		,
	Q_bOP=> 				, 
	Q_bCom=> 				, 
	Q_bError=> 				,
	Q_sState=>				);
	
(*///////////////////////////////////////////////////////////*)
(*	Device States *)
CASE fbUniHBComOperator.Q_EState OF
(*///////////////////////////////////////////////////////////*)
E_HB_Device_Init:
		bEventStartupDone := FALSE;
		Q_stOutput.sState 		:=	CONCAT(I_stInput.sName,'| ');
		Q_stOutput.sState		:=	CONCAT(Q_stOutput.sState, fbUniHBComOperator.Q_sState);
		
E_HB_Device_CheckID,
E_HB_Device_EventStartup:	
		ac00_Event();
		bResetDone := FALSE;
		bStartupDone := FALSE;
		iStepSet := 0;
		Q_stOutput.sState 		:=	CONCAT(I_stInput.sName,'| ');
		Q_stOutput.sState		:=	CONCAT(Q_stOutput.sState, fbUniHBComOperator.Q_sState);
(*///////////////////////////////////////////////////////////*)
E_HB_Device_Reset:
		ac00_Event();
		ac01_SetReset();
		
		Q_stOutput.sState 		:=	CONCAT(I_stInput.sName,'| ');
		Q_stOutput.sState		:=	CONCAT(Q_stOutput.sState, fbUniHBComOperator.Q_sState);
		Q_stOutput.sState		:=	CONCAT(Q_stOutput.sState, '| ');
		Q_stOutput.sState		:=	CONCAT(Q_stOutput.sState, sStateReset);
(*///////////////////////////////////////////////////////////*)
E_HB_Device_WaitCom:
		ac00_Event();
		iStepSet := 0;
		Q_stOutput.sState 		:=	CONCAT(I_stInput.sName,'| ');
		Q_stOutput.sState		:=	CONCAT(Q_stOutput.sState, fbUniHBComOperator.Q_sState);
(*///////////////////////////////////////////////////////////*)		
E_HB_Device_Startup:
		ac00_Event();
		ac01_SetLED();	
		
		Q_stOutput.sState 		:=	CONCAT(I_stInput.sName,'| ');
		Q_stOutput.sState		:=	CONCAT(Q_stOutput.sState, fbUniHBComOperator.Q_sState);
(*///////////////////////////////////////////////////////////*)
E_HB_Device_OP:
		ac00_Event();
		ac01_SetLED();	
		ac10_Counter();
		
		Q_stOutput.sState 		:=	CONCAT(I_stInput.sName,'| ');
		Q_stOutput.sState		:=	CONCAT(Q_stOutput.sState, fbUniHBComOperator.Q_sState);
END_CASE

(*///////////////////////////////////////////////////////////*)
(* Sendebaustein *)
IF fbUniHBComOperator.Q_bActivateSend
THEN
	Q_sFiFoSend :=	sFiFoSend;
END_IF
	
(*///////////////////////////////////////////////////////////*)
(* Outputs *)
Q_stOutput.bCOM 		:=	fbUniHBComOperator.Q_bCom;
Q_stOutput.bError 		:= 	fbUniHBComOperator.Q_bError;
Q_stOutput.bStartupDone	:=	fbUniHBComOperator.Q_bOP;
Q_stOutput.dwChanges	:=	fbUniHBComOperator.Q_dwChanges;

ACTION ac00_Event:
(*============================================================================================*)
(*	EVENT Schrittkette *)
(*============================================================================================*)

IF fbUniHBComOperator.Q_bResetEvents
THEN
	sReceived := '';
	
	(* Ausgänge alle auf 0 setzen *)
	FOR i := 1 TO 6 BY 1 DO 		
		iDimmMem[i] := 0;
		Q_stOutput.bButtons[i] := FALSE;
	END_FOR
	
	Q_stOutput.lrTemp := 0;
	Q_stOutput.lrBrs := 0;
	Q_stOutput.lrRhd := 0;	
ELSE
	sReceived := I_StringReceived;
END_IF
(*
fbBusTasterEvent(
	I_bExecute			:=	fbUniHBComOperator.Q_bExecuteEvents,
	I_bReset			:=	fbUniHBComOperator.Q_bResetEvents,
	I_bFaultDetection	:=	bInputFaultDetect,
	I_tFaultDetectTime	:=	tInputFaultDetect,
	I_sID				:= 	DINT_TO_STRING(I_stInput.diID), 
	I_sInstID			:= 	INT_TO_STRING(16), 
	I_sReceivedString	:= 	sReceived, 
	Q_bOut				=> 	Q_stOutput.bButtons);*)

fbBusTasterEvent(
	I_bExecute			:=	fbUniHBComOperator.Q_bExecuteEvents,
	I_bReset			:=	fbUniHBComOperator.Q_bResetEvents,
	I_diID				:= 	I_stInput.diID, 
	I_iInstID			:= 	16, 
	I_sReceivedString	:= 	sReceived, 
	I_bFaultDetection	:=	bInputFaultDetect,
	I_tFaultDetectTime	:=	tInputFaultDetect,
	Q_bOut				=> Q_stOutput.bButtons, 
	Q_bStartupDone		=> 	);	
	
IF I_stInput.bExtInputs	(* Externe Eingänge Aktivieren *)
THEN
		
	fbBusTasterEventExt(
		I_bExecute			:=	fbUniHBComOperator.Q_bExecuteEvents,
		I_bReset			:=	fbUniHBComOperator.Q_bResetEvents,
		I_diID				:= 	I_stInput.diID, 
		I_iInstID			:= 	32, 
		I_sReceivedString	:= 	sReceived, 
		I_bFaultDetection	:=	FALSE,
		I_tFaultDetectTime	:=	tInputFaultDetect,
		Q_bOut				=>  Q_stOutput.bButtonsExt, 
		Q_bStartupDone		=> 	);	
END_IF

fbBusTempEvent(
	I_bExecute 				:=	fbUniHBComOperator.Q_bExecuteEvents,
	I_bReset				:=	fbUniHBComOperator.Q_bResetEvents,
	I_diID					:= 	I_stInput.diID, 
	I_iInstID				:= 	1, 
	I_sReceivedString		:= 	sReceived, 
	Q_lrTemp				=> 	Q_stOutput.lrTemp,
	Q_tUpdate				=>	Q_stOutput.tLastUpdateTemp,
	Q_sLastUpdate			=>	Q_stOutput.sLastUpdateTemp);
	
fbBusBrsEvent(
	I_bExecute 				:=	fbUniHBComOperator.Q_bExecuteEvents,
	I_bReset				:=	fbUniHBComOperator.Q_bResetEvents,
	I_diID					:= 	I_stInput.diID, 
	I_iInstID				:= 	1, 
	I_sReceivedString		:= 	sReceived, 
	Q_lrBrs					=> 	Q_stOutput.lrBrs,
	Q_tUpdate				=>	Q_stOutput.tLastUpdateBrs,
	Q_sLastUpdate			=>	Q_stOutput.sLastUpdateBrs);
	
fbBusRhdEvent(
	I_bExecute 				:=	fbUniHBComOperator.Q_bExecuteEvents,
	I_bReset				:=	fbUniHBComOperator.Q_bResetEvents,
	I_diID					:= 	I_stInput.diID, 
	I_iInstID				:= 	1, 
	I_sReceivedString		:= 	sReceived, 
	Q_lrRhd					=> 	Q_stOutput.lrRhd,
	Q_tUpdate				=>	Q_stOutput.tLastUpdateRhd,
	Q_sLastUpdate			=>	Q_stOutput.sLastUpdateRhd);
	
fbBusPingEvent(
	I_bExecute 				:=	fbUniHBComOperator.Q_bExecuteEvents,
	I_bReset				:=	fbUniHBComOperator.Q_bResetEvents,
	I_diID					:= 	I_stInput.diID, 
	I_sReceivedString		:= 	sReceived, 
	Q_bOut					=> 	);
	
bEventStartupDone :=	fbBusTasterEvent.Q_bStartupDone
						AND (fbBusTasterEventExt.Q_bStartupDone
							OR NOT I_stInput.bExtInputs)
						AND fbBusTempEvent.Q_bStartupDone
						AND fbBusBrsEvent.Q_bStartupDone
						AND fbBusRhdEvent.Q_bStartupDone
						AND fbBusPingEvent.Q_bStartupDone;
END_ACTION

ACTION ac01_SetLED:
(*============================================================================================*)
(*	LED Helligkeit Setzen/ Startup Schrittkette *)
(*============================================================================================*)

(* Selbstcheck- Eingänge automatisch prüfen *)

tSelfCheckStatus := I_tSelfCheckTime;

tonStepStartup();
tonSelfCheck(
	IN := iStepSet = 0
			AND NOT bSendeAnforderung
			AND NOT bSendeAnforderungExt
			AND NOT bSendeAnforderungBG
			AND NOT fbUniHBComOperator.Q_bStartupStart
			AND I_bSelfCheckAuto,
	PT := tSelfCheckStatus);

IF (tonSelfCheck.Q
	AND I_bSelfCheckAuto)
	OR (NOT tonSelfCheck.Q
	AND I_bSelfCheck)
	AND NOT bGlobalPingActive (* Achtung Globale Vaariable, Wenn Ping aktiv ist *)
THEN
	bSelfCheckAnforderung := TRUE;
END_IF
	
(*setzen der LED Helligkeiten (0-100 Prozent *)
(* Neu, es werden alle LEDs zu einem String zusammengefügt und Gleichzeitig gesetzt *)
cntchangesDimm := 0;
cntChangesDimmExt :=0;
	
FOR l := 1 TO 6 BY 1 DO
	IF iDimmMem[l] <> I_stInput.iLED[l]
	THEN
		cntChangesDimm := cntChangesDimm +1;
	END_IF

	IF  iDimmMemExt[l]<> I_stInput.iLEDExt[l]
	THEN
		cntChangesDimmExt := cntChangesDimmExt +1;
	END_IF
END_FOR

CASE iStepSet OF
(*============================================================================================*)
0:	(* INIT und warten auf Change *)
	tonStepStartup.PT:= tStartupLEDOn;				
	tonStepStartup.IN := FALSE; 
	sFiFoSend := ''; 
	
	fbRS485HBStringBuilder(
		I_bExecute:= 		FALSE );
		
	(* Änderungs- Anforderungen Prüfen*)
	FOR e := 1 TO 6 BY 1 DO
		IF cntChangesDimm<>0
		THEN
			(* Helligkeitanforderung Interne LEDs speichern *)
			bSendeAnforderung := TRUE;
			iDimmAnf[e] 	:= I_stInput.iLED[e];
		END_IF
		
		IF cntChangesDimmExt <> 0
		THEN
			(* Helligkeitanforderung Externe LEDs speichern *)
			bSendeAnforderungExt := TRUE;
			iDimmAnfExt[e] 	:= I_stInput.iLEDExt[e];
		END_IF
		
		IF I_stInput.iLEDBg <>iDimmBgMem
		THEN
			(* Helligkeitsanforderung Hintergrundbeleuchtung *)
			bSendeAnforderungBG := TRUE;
			iDimmBGAnf		:= I_stInput.iLEDBg;
		END_IF
	END_FOR
	
	(* Reagieren auf Anforderungen *)
	IF ((bSendeAnforderung
		OR bSendeAnforderungExt
		OR bSendeAnforderungBG)
		AND bSetExecute)
		AND NOT fbUniHBComOperator.Q_bStartupStart
		AND NOT bSelfCheckAnforderung
	THEN
		(* Helligkeitsvorgaben speichern in Mem Arrays *)
		FOR h := 1 TO 6 BY 1 DO
			iDimmMem[h] := I_stInput.iLED[h];
			iDimmMemExt[h] := I_stInput.iLEDExt[h];
			iDimmBgMem := I_stInput.iLEDBg;
		END_FOR
		
		iStepSet := 10;
	ELSIF
		fbUniHBComOperator.Q_bStartupStart
	THEN
		bStartupDone := FALSE;
		iStepSet := 100;	(* Startup *)
	ELSIF
		bSelfCheckAnforderung
	THEN
		iStepSet := 122; 	(* Eingänge abfragen Selbsttest *)
	END_IF
	
(*============================================================================================*)
10:	(* Prüfen welche Anforderung ausgeführt werden soll *)	
	IF	bSendeAnforderungBG
		AND NOT bSendeAnforderung
		AND NOT bSendeAnforderungExt 
	THEN
		iStepSet := 22;(* Direkt nur die Hintergrund Helligkeit setzen *)
	ELSE
		(* Nur Interne LEDs Schreiben *)
		IF bSendeAnforderung
			AND NOT bSendeAnforderungExt
			AND NOT bSendeAnforderungBG
		THEN
			FOR e := 1 TO 6 BY 1 DO
				fbRS485HBStringBuilder.I_iP1[e] :=iDimmAnf[e];
			END_FOR
	
			fbRS485HBStringBuilder(
				I_bExecute:= 		TRUE, 
				I_diID:= 			I_stInput.diID, 
				I_iInstID:= 		49, 
				I_EnumHBUnitTX:= 	E_EnumHBUnitTX.E_HB_UNIT_LED, 
				I_EnumHBCmdTX:= 	E_EnumHBCmdTX.E_HB_CMD_ON, 
				I_iCnt:= 			6,  
				Q_sOut=> 			sSendString);
				
			(* Senden an FiFo*)
			IF I_bFiFoDone
				AND fbRS485HBStringBuilder.Q_bDone
			THEN
				sFiFoSend :=	sSendString;
			END_IF
			
			IF NOT I_bFiFoDone
			THEN
				fbRS485HBStringBuilder(
					I_bExecute:= 		FALSE );
					
				bSendeAnforderung := FALSE;
				sLastSendString :=	sFiFoSend;
				iStepSet := 20;
			END_IF
		ELSIF
			(* Nur Externe LEDs Schreiben *)	
			bSendeAnforderungExt
			AND NOT bSendeAnforderung
			AND NOT bSendeAnforderungBG
		THEN
			FOR e := 1 TO 6 BY 1 DO
				fbRS485HBStringBuilder.I_iP1[e] :=iDimmAnfExt[e];
			END_FOR
			
			fbRS485HBStringBuilder(
				I_bExecute:= 		TRUE, 
				I_diID:= 			I_stInput.diID, 
				I_iInstID:= 		65, 
				I_EnumHBUnitTX:= 	E_EnumHBUnitTX.E_HB_UNIT_LED, 
				I_EnumHBCmdTX:= 	E_EnumHBCmdTX.E_HB_CMD_ON, 
				I_iCnt:= 			6, 
				Q_sOut=> 			sSendString);
			
			(* Senden an FiFo*)
			IF I_bFiFoDone
			THEN
				sFiFoSend :=	sSendString;
			END_IF
			
			IF NOT I_bFiFoDone
			THEN
				fbRS485HBStringBuilder(
					I_bExecute:= 		FALSE );
					
				bSendeAnforderungExt := FALSE;
				sLastSendString :=	sFiFoSend;
				iStepSet := 20;
			END_IF
		ELSE
			(* Externe und Interne LEDs Schreiben *)
			bMemExt := TRUE; (* Speichern, damit anschließend noch die Externen LEDs gesetzt werden *)
			
			FOR e := 1 TO 6 BY 1 DO
				fbRS485HBStringBuilder.I_iP1[e] :=iDimmAnf[e];
			END_FOR
			
			fbRS485HBStringBuilder(
				I_bExecute:= 		TRUE, 
				I_diID:= 			I_stInput.diID, 
				I_iInstID:= 		49, 
				I_EnumHBUnitTX:= 	E_EnumHBUnitTX.E_HB_UNIT_LED, 
				I_EnumHBCmdTX:= 	E_EnumHBCmdTX.E_HB_CMD_ON, 
				I_iCnt:= 			6,  
				Q_sOut=> 			sSendString);
			
			(* Senden an FiFo*)
			IF I_bFiFoDone
			THEN
				sFiFoSend :=	sSendString;
			END_IF
			IF NOT I_bFiFoDone
			THEN
				fbRS485HBStringBuilder(
					I_bExecute:= 		FALSE );
					
				bSendeAnforderung := FALSE;
				bSendeAnforderungExt := FALSE;
				sLastSendString :=	sFiFoSend;
				iStepSet := 20;
			END_IF
		END_IF
	END_IF
(*============================================================================================*)	
20:	(* Warten bis nicht Busy *)	
	
	IF I_bFiFoDone
	THEN
		sFiFoSend := ''; 
		IF NOT bMemExt
		THEN
			IF bSendeAnforderungBG
			THEN
				iStepSet := 22;
			ELSE
				iStepSet := 0;
			END_IF
		ELSE
			iStepSet :=	21;
		END_IF
	END_IF
	
(*============================================================================================*)	
21:	(* Externe LEDs Senden *)	
	bMemExt := FALSE;
	bSendeAnforderungExt := FALSE;
	
	FOR e := 1 TO 6 BY 1 DO
		fbRS485HBStringBuilder.I_iP1[e] :=iDimmAnfExt[e];
	END_FOR
	
	fbRS485HBStringBuilder(
		I_bExecute:= 		TRUE, 
		I_diID:= 			I_stInput.diID, 
		I_iInstID:= 		65, 
		I_EnumHBUnitTX:= 	E_EnumHBUnitTX.E_HB_UNIT_LED, 
		I_EnumHBCmdTX:= 	E_EnumHBCmdTX.E_HB_CMD_ON, 
		I_iCnt:= 			6, 
		Q_sOut=> 			sSendString);
		
	(* Senden an FiFo*)
	IF I_bFiFoDone
	THEN
		sFiFoSend :=	sSendString;
	END_IF
	IF NOT I_bFiFoDone
	THEN
		fbRS485HBStringBuilder(
			I_bExecute:= 		FALSE );
					
		sLastSendString :=	sFiFoSend;
		iStepSet := 20;
	END_IF
	
(*============================================================================================*)	
22:	(* Hintergrundbeleuchtung senden *)		
	bSendeAnforderungBG := FALSE;
	
	fbRS485HBStringBuilder.I_iP1[1]:= iDimmBGAnf;
	
	fbRS485HBStringBuilder(
		I_bExecute:= 		TRUE, 
		I_diID:= 			I_stInput.diID, 
		I_iInstID:= 		16, 
		I_EnumHBUnitTX:= 	E_EnumHBUnitTX.E_HB_UNIT_LBN, 
		I_EnumHBCmdTX:= 	E_EnumHBCmdTX.E_HB_CMD_SET_MBR, 
		I_iCnt:= 			1, 
		Q_sOut=> 			sSendString);
		
	(* Senden an FiFo*)
	IF I_bFiFoDone
	THEN
		sFiFoSend :=	sSendString;
	END_IF
	IF NOT I_bFiFoDone
	THEN
		fbRS485HBStringBuilder(
			I_bExecute:= 		FALSE );
			
		sLastSendString :=	sFiFoSend;
		iStepSet := 20;
	END_IF

(*============================================================================================*)	
(* Startup LEDS einmal Einschalten *)
100:	
	tonStepStartup.PT:= tStartupLEDOn;
	tonStepStartup.IN := TRUE;
	
	IF tonStepStartup.Q
	THEN
		iStepSet := 110;
	END_IF
	
(*============================================================================================*)
110:	(* String senden *)	
	tonStepStartup.IN := FALSE;
	
	fbRS485HBStringBuilder.I_iP1[1]:= 100;
	
	fbRS485HBStringBuilder(
		I_bExecute:= 		TRUE, 
		I_diID:= 			I_stInput.diID, 
		I_iInstID:= 		16, 
		I_EnumHBUnitTX:= 	E_EnumHBUnitTX.E_HB_UNIT_LBN, 
		I_EnumHBCmdTX:= 	E_EnumHBCmdTX.E_HB_CMD_SET_MBR, 
		I_iCnt:= 			1, 
		Q_sOut=> 			sSendString);
			
	(* Senden an FiFo*)
	IF I_bFiFoDone
	THEN
		sFiFoSend :=	sSendString;
	END_IF
	IF NOT I_bFiFoDone
	THEN
		fbRS485HBStringBuilder(
			I_bExecute:= 		FALSE );
			
		iStepSet := 111;
	END_IF
	
(*============================================================================================*)	
111:(* Warten bis nicht Busy *)	
	IF I_bFiFoDone
	THEN
		sFiFoSend := ''; 
		tonStepStartup.IN := TRUE;
		
		IF tonStepStartup.Q
		THEN
			tonStepStartup.IN := FALSE;
			iStepSet := 120;
		END_IF
	END_IF
	
(*============================================================================================*)
120:	(* String senden *)	

	fbRS485HBStringBuilder.I_iP1[1]:= 0;
	
	fbRS485HBStringBuilder(
		I_bExecute:= 		TRUE, 
		I_diID:= 			I_stInput.diID, 
		I_iInstID:= 		16, 
		I_EnumHBUnitTX:= 	E_EnumHBUnitTX.E_HB_UNIT_LBN, 
		I_EnumHBCmdTX:= 	E_EnumHBCmdTX.E_HB_CMD_SET_MBR, 
		I_iCnt:= 			1, 
		Q_sOut=> 			sSendString);
			
	(* Senden an FiFo*)
	IF I_bFiFoDone
	THEN
		sFiFoSend :=	sSendString;
	END_IF
	IF NOT I_bFiFoDone
	THEN
		fbRS485HBStringBuilder(
			I_bExecute:= 		FALSE );
			
		iStepSet := 121;
	END_IF

(*============================================================================================*)	
121:(* Warten bis nicht Busy *)	
	tonStepStartup.PT:= T#500MS;
	
	IF I_bFiFoDone
	THEN
		sFiFoSend := ''; 
		tonStepStartup.IN := TRUE;
		
		IF tonStepStartup.Q
		THEN
			tonStepStartup.IN := FALSE;
			iStepSet := 122;
		END_IF
	END_IF
	
(*============================================================================================*)
122:(* Eingangsstatus abfragen  Intern senden *)	
	fbRS485HBStringBuilder.I_iP1[1]:= 0;
	
	fbRS485HBStringBuilder(
		I_bExecute:= 		TRUE, 
		I_diID:= 			I_stInput.diID, 
		I_iInstID:= 		16, 
		I_EnumHBUnitTX:= 	E_EnumHBUnitTX.E_HB_UNIT_BTN, 
		I_EnumHBCmdTX:= 	E_EnumHBCmdTX.E_HB_CMD_gSTATUS, 
		I_iCnt:= 			6, 
		Q_sOut=> 			sSendString);
			
	(* Senden an FiFo*)
	IF I_bFiFoDone
	THEN
		sFiFoSend :=	sSendString;
	END_IF
	IF NOT I_bFiFoDone
	THEN
		fbRS485HBStringBuilder(
			I_bExecute:= 		FALSE );
			
		iStepSet := 123;
	END_IF

(*============================================================================================*)	
123:(* Warten bis nicht Busy *)	
	IF I_bFiFoDone
	THEN
		sFiFoSend := ''; 
		
		IF bSelfCheckAnforderung
		THEN
			tonStepStartup.PT:= T#20MS;
			tonStepStartup.IN := TRUE;
			
			IF I_stInput.bExtInputs
			THEN
				IF tonStepStartup.Q
				THEN
					tonStepStartup.IN := FALSE;
					iStepSet := 124;
				END_IF
			ELSE
				tonStepStartup.IN := FALSE;
				iStepSet := 130;
			END_IF
		ELSE
			
			tonStepStartup.IN := TRUE;
			IF tonStepStartup.Q
			THEN
				tonStepStartup.IN := FALSE;
				iStepSet := 124;
			END_IF
		END_IF
	END_IF
	
(*============================================================================================*)
124:	(* Eingangsstatus abfragen  Extern senden *)	

	fbRS485HBStringBuilder.I_iP1[1]:= 0;
	
	fbRS485HBStringBuilder(
		I_bExecute:= 		TRUE, 
		I_diID:= 			I_stInput.diID, 
		I_iInstID:= 		32, 
		I_EnumHBUnitTX:= 	E_EnumHBUnitTX.E_HB_UNIT_BTN, 
		I_EnumHBCmdTX:= 	E_EnumHBCmdTX.E_HB_CMD_gSTATUS, 
		I_iCnt:= 			6, 
		Q_sOut=> 			sSendString);
			
	(* Senden an FiFo*)
	IF I_bFiFoDone
	THEN
		sFiFoSend :=	sSendString;
	END_IF
	IF NOT I_bFiFoDone
	THEN
		fbRS485HBStringBuilder(
			I_bExecute:= 		FALSE );
			
		iStepSet := 130;
	END_IF
	
(*============================================================================================*)	
130:(* Warten bis nicht Busy *)	
	IF I_bFiFoDone
	THEN
		sFiFoSend := ''; 
		
		IF bSelfCheckAnforderung
			AND NOT I_bSelfCheck
		THEN
			bSelfCheckAnforderung := FALSE;
			iStepSet := 0;
		ELSE
			tonStepStartup.IN := TRUE;
			IF tonStepStartup.Q
			THEN
				bStartupDone := TRUE;
				tonStepStartup.IN := FALSE;
				iStepSet := 10;	(* Anschließend noch einmal die Eingangs Helligkeit setzen *)
			END_IF
		END_IF
	END_IF	

END_CASE

(*bErrorSet := fbRS485SendCmd.Q_bError;*)
END_ACTION

ACTION ac01_SetReset:
(*============================================================================================*)
(*	RESET Schrittkette *)
(*============================================================================================*)
tonResetTimeout(
	PT := tResetTimeout);

(* Einfaches Setzen der LED Helligkeiten (0-100 Prozent *)
CASE iStepSet OF
(*============================================================================================*)
0:	sStateReset 		:= 'INIT';
	
	fbRS485HBStringBuilder(
		I_bExecute:= 		FALSE );
		
	IF fbUniHBComOperator.Q_bSendResetCmd
	THEN
	
		sFiFoSend 			:= ''; 
		bResetDone 			:= FALSE;
		tonResetTimeout.IN 	:= FALSE;
				
		iStepSet := iStepSet +1;
	END_IF

(*============================================================================================*)	
1:	sStateReset := 'Sende Reset Befehl';
	bResetBusy := TRUE;
	bErrorReset := FALSE;
	
	fbRS485HBStringBuilder(
		I_bExecute:= 		TRUE, 
		I_diID:= 			I_stInput.diID, 
		I_iInstID:= 		1, 
		I_EnumHBUnitTX:= 	E_EnumHBUnitTX.E_HB_UNIT_SYS, 
		I_EnumHBCmdTX:= 	E_EnumHBCmdTX.E_HB_CMD_RESET, 
		I_iCnt:= 			1, 
		Q_sOut=> 			sSendString);

	(* Senden an FiFo*)
	IF I_bFiFoDone
	THEN
		sFiFoSend :=	sSendString;
	END_IF
	
	IF NOT I_bFiFoDone
	THEN
		fbRS485HBStringBuilder(
			I_bExecute:= 		FALSE );
		
		iStepSet := iStepSet+1;
	END_IF

(*============================================================================================*)
2:	sStateReset := 'Sende Reset Befehl';

	IF I_bFiFoDone
	THEN
		sFiFoSend := ''; 
		iStepSet := iStepSet+1;
	END_IF
	
(*============================================================================================*)	
3:	sStateReset := 'Reset durchgeführt, Warte auf Ping';
	bResetDone := TRUE;
	bResetBusy := FALSE;
	
END_CASE
END_ACTION

ACTION ac10_Counter:
(*============================================================================================*)
(* 	Zähler *)
(*============================================================================================*)
FOR j := 1 TO 6 BY 1 DO 
	r_TrigCountBtn[j](
		CLK := Q_stOutput.bButtons[j]);
		
	IF r_TrigCountBtn[j].Q
	THEN
		Q_stCnt.dwCntButtons[j] := Q_stCnt.dwCntButtons[j]+1;
	END_IF
	
END_FOR
END_ACTION

ACTION ac99_Doku:
(*======================================================================================================================================*)
(*	DOKU	*)
(*======================================================================================================================================*)
(* Wichtiger Hinweis:
		-Bei dem 6 Fach Taster ist zu Beachten, dass es nur 4 Externe EA/s gibt also 4 LEDs und 4 Taster, 
		da der ESP 32 Nur 10Es und 10As besitzt.
		- Die 4 Zusätzlichen Ausgänge werden von der Hintergrundbeleuchtung Ausgeschlossen und müssen über den Befehl: SET_MBR einzeln 
			gesetzt werden! *)	
	
(* Verdrahtung:		
	Verdrahtung füR: KL6041
        +-------+
        |       |
        | TxD+ ----+
        |         |----> RS485 A (zum Bus)
        | RxD+ ----+
        |         |
        | TxD− ----+
        |         |----> RS485 B (zum Bus)
        | RxD− ----+
        +-------+	*)
		
(*======================================================================================================================================*)
(* Telegrammbeschreibung *)

(*	Die XML Dateien der verschiedenen Module sind grundsätzlich immer gleich aufgebaut. 
	Je Instanz der verschiedenen Sensoren und Aktoren werden die zu sendenden Befehle bzw. 
	die zu empfangenen Events beschrieben. 
	Alle Telegramme sind ASCII kodiert und sind umgeben mit dem binären Startzeichen 0xFD und dem binären Endezeichen 0xFE.

	Grundaufbauer aller im Folgenden beschriebenen Telegramme:
	
	-Startzeichen immer 0xFD.
	-Punkte dienen als Trennzeichen der verschiedenen Elemente
	-Endezeichen immer 0xFE.
	-Element 1 ist die Geräte-ID, die entsprechend der verwendeten Module angepasst werden muss (hier beispielhaft jeweils 12345)
	-Element 2 ist ein Schlüsselwort für den jeweiligen Funktionstyp (z.b. BTN, LED, DIM, usw)
	-Element 3 ist die InstanzID gemäß XML Templates (also welche Taster oder welcher Dimmer konkret gemeint ist)
	-Element 4 zeigt die jeweilige Aktion zum Funktionstypen (z.b. ON, OFF, STATUS)
	-Anschließend kommen optional diverse Parameter, die mit P1,P2,...P3 bezeichnet werden
	
	Im Folgenden wird nur noch auf die speziellen Telegramdaten eingegangen:
	
	(*------------------------------------------------------------*)
	Taster oder digitaler Eingang (Sensor):
	(*------------------------------------------------------------*)
	Telegram Event:  	
	
	\xFD 12345.BTN.17.STATUS.P1 \xFE
	
		Funktionstyp:		BTN (kurz für Button)
		Instanz-ID:			hier 17 (in XML nachschauen)
		Aktion:				STATUS
		P1:					1, wenn Taste gedrückt bzw. Eingang aktiv
							0, wenn Taste losgelassen bzw. Eingang inaktiv
	
	Telegram Statusabfrage:  	
	
	\xFD 12345.BTN.17.gSTATUS \xFE
	
		Antwort:  			\xFD 12345.BTN.17.rSTATUS.P1 \xFE
		P1:					1, wenn Taste gedrückt bzw. Eingang aktiv
							0, wenn Taste losgelassen bzw. Eingang inaktiv

	(*------------------------------------------------------------*)
	Led (Aktor):
	(*------------------------------------------------------------*)
	Telegram Helligkeit setzen:  	
	
	\xFD 12345.LED.50.ON.P1.P2.P3 \xFE
	
		Funktionstyp:			LED
		Instanz-ID:				hier 50 (in XML nachschauen)
		Aktion:					ON
		P1:						gewünschte Helligkeit 0-100
		P2:						Einschaltdauer in 100stel Sekunden (0 = daueran)
		P3:						Einschaltverzögerung in Sekunden (0 = ohne Verzögerung)
	
	Telegram Mindesthelligkeit:  	
	
	\xFD 12345.LED.50.SET_MBR.P1 \xFE
		
		Aktion:					SET_MBR (Setzt eine Mindesthelligkeit, die auch dann erhalten bleibt, wenn man per OFF ausschaltet)
		P1:						gewünschte Helligkeit 0-100
	
	Telegram Statusabfrage:  	

	\xFD 12345.LED.50.gSTATUS \xFE
	
		Antwort:  				\xFD 12345.LED.50.rSTATUS.P1.P2 \xFE
		P1:						aktuelle Helligkeit 0-100
		P2:						Einschaltdauer in 100stel Sekunden
	
	(*------------------------------------------------------------*)
	Hintergrundbeleuchtung (Aktor):
	(*------------------------------------------------------------*)
	Telegram Minhelligkeit:  
	
	\xFD 12345.LBN.16.SET_MBR.P1 \xFE
	
		Aktion:					SET_MBR ((Setzt eine Mindesthelligkeit, die auch dann erhalten bleibt, wenn man per OFF ausschaltet)
		P1:						gewünschte Helligkeit 0-100
		
	Telegram Statusabfrage:  	

	\xFD 12345.LBN.16.gSTATUS \xFE
	
		Antwort:  				\xFD 12345.LBN.16.rSTATUS.P1 \xFE
		P1:						aktuelle Helligkeit 0-100

	(*------------------------------------------------------------*)
	Temperatursensor (Sensor):
	(*------------------------------------------------------------*)
	Telegram Event:  	
	
	\xFD 12345.TMP.1.STATUS.P1.P2 \xFE
	
		Funktionstyp:			TMP (kurz für Temperatur)
		Instanz-ID:				hier 1 (in XML nachschauen)
		Aktion:					STATUS
		P1:						Temperatur in Grad Vorkommastellen
		P2:						Temperatur in Grad Nachkommastellen
	
	Telegram Statusabfrage:  
	
	\xFD 12345.TMP.1.gSTATUS \xFE
	
		Antwort:  				\xFD 12345.TMP.1.rSTATUS.P1.P2 \xFE
		P1:						Temperatur in Grad Vorkommastellen
		P2:						Temperatur in Grad Nachkommastellen

	(*------------------------------------------------------------*)
	Feuchtesensor (Sensor):
	(*------------------------------------------------------------*)
	Telegram Event:  	

	\xFD 12345.RHD.1.STATUS.P1.P2 \xFE
	
		Funktionstyp:			RHD (kurz für Relative Humidity)
		Instanz-ID:				hier 1 (in XML nachschauen)
		Aktion:					STATUS
		P1:						Relative Luftfeuchtigkeit 0-100 Vorkommastellen
		P2:						Relative Luftfeuchtigkeit 0-100 Nachkommastellen

	Telegram Statusabfrage:  	
	
	\xFD 12345.RHD.1.gSTATUS \xFE
	
	Antwort:  					\xFD 12345.RHD.1.rSTATUS.P1 \xFE
	P1:							Relative Luftfeuchtigkeit 0-100 Vorkommastellen
	P2:							Relative Luftfeuchtigkeit 0-100 Nachkommastellen

	(*------------------------------------------------------------*)
	Helligkeitssensor (Sensor):
	(*------------------------------------------------------------*)
	Telegram Event:  	
	
	\xFD 12345.BRS.23.STATUS.P1.P2 \xFE
	
		Funktionstyp:			BRS (kurz für Brightness Sensor)
		Instanz-ID:				hier 23 (in XML nachschauen)
		Aktion:					STATUS
		P1:						Relative Helligkeit 0-255 Vorkommastellen
		P2:						Relative Helligkeit 0-255 Nachkommastellen
	
	Telegram Statusabfrage:  	
	
	\xFD 12345.BRS.23.gSTATUS \xFE
	
	Antwort:  					\xFD 12345.BRS.23.rSTATUS.P1 \xFE
	P1:							Relative Helligkeit 0-255 Vorkommastellen
	P2:							Relative Helligkeit 0-255 Nachkommastellen

(*======================================================================================================================================*)
(* Alle Telegramme im Überblick *)	

	<?xml version="1.0" encoding="utf-8"?>
	<Comm Title="Haus-Bus ID 12345" Comment="" Baudrate="57600" Databits="8" Parity="1" EndChar="510">
	<CommCmd Title="6-fach Taster 12345 - Hintergrundbeleuchtung" Comment="" CmdOn="\xFD12345.LBN.16.SET_MBR.&lt;v&gt;.0\xFE" CmdOff="\xFD12345.LBN.16.SET_MBR.0\xFE" Unit="" Analog="true" Text="false" Sensor="false" SourceValHigh="100" DestValHigh="100"/>
	<CommCmd Title="6-fach Taster 12345 - Temperatursensor" Comment="" CmdOn="\xFD12345.TMP.1.STATUS.\v\xFE" CmdOff="" Unit="&lt;v.2&gt;" Analog="true" Text="false" Sensor="true" SourceValHigh="100" DestValHigh="100"/>
	<CommCmd Title="6-fach Taster 12345 - Feuchtesensor" Comment="" CmdOn="\xFD12345.RHD.1.STATUS.\v\xFE" CmdOff="" Unit="&lt;v.x&gt;" Analog="true" Text="false" Sensor="true" SourceValHigh="100" DestValHigh="100"/>
	<CommCmd Title="6-fach Taster 12345 - Helligkeitssensor" Comment="" CmdOn="\xFD12345.BRS.1.STATUS.\v\xFE" CmdOff="" Unit="&lt;v.x&gt;" Analog="true" Text="false" Sensor="true" SourceValHigh="100" DestValHigh="100"/>
	<CommCmd Title="6-fach Taster 12345 - Led 1" Comment="" CmdOn="\xFD12345.LED.49.ON.&lt;v&gt;.0\xFE" CmdOff="\xFD12345.LED.49.OFF\xFE" Unit="" Analog="true" Text="false" Sensor="false" SourceValHigh="100" DestValHigh="100"/>
	<CommCmd Title="6-fach Taster 12345 - Led 2" Comment="" CmdOn="\xFD12345.LED.50.ON.&lt;v&gt;.0\xFE" CmdOff="\xFD12345.LED.50.OFF\xFE" Unit="" Analog="true" Text="false" Sensor="false" SourceValHigh="100" DestValHigh="100"/>
	<CommCmd Title="6-fach Taster 12345 - Led 3" Comment="" CmdOn="\xFD12345.LED.51.ON.&lt;v&gt;.0\xFE" CmdOff="\xFD12345.LED.51.OFF\xFE" Unit="" Analog="true" Text="false" Sensor="false" SourceValHigh="100" DestValHigh="100"/>
	<CommCmd Title="6-fach Taster 12345 - Led 4" Comment="" CmdOn="\xFD12345.LED.52.ON.&lt;v&gt;.0\xFE" CmdOff="\xFD12345.LED.52.OFF\xFE" Unit="" Analog="true" Text="false" Sensor="false" SourceValHigh="100" DestValHigh="100"/>
	<CommCmd Title="6-fach Taster 12345 - Led 5" Comment="" CmdOn="\xFD12345.LED.53.ON.&lt;v&gt;.0\xFE" CmdOff="\xFD12345.LED.53.OFF\xFE" Unit="" Analog="true" Text="false" Sensor="false" SourceValHigh="100" DestValHigh="100"/>
	<CommCmd Title="6-fach Taster 12345 - Led 6" Comment="" CmdOn="\xFD12345.LED.54.ON.&lt;v&gt;.0\xFE" CmdOff="\xFD12345.LED.54.OFF\xFE" Unit="" Analog="true" Text="false" Sensor="false" SourceValHigh="100" DestValHigh="100"/>
	<CommCmd Title="6-fach Taster 12345 - Taster 1" Comment="" CmdOn="\xFD12345.BTN.17.STATUS.\v\xFE" CmdOff="" Unit="&lt;v.x&gt;" Analog="true" Text="false" Sensor="true" SourceValHigh="100" DestValHigh="100"/>
	<CommCmd Title="6-fach Taster 12345 - Taster 2" Comment="" CmdOn="\xFD12345.BTN.18.STATUS.\v\xFE" CmdOff="" Unit="&lt;v.x&gt;" Analog="true" Text="false" Sensor="true" SourceValHigh="100" DestValHigh="100"/>
	<CommCmd Title="6-fach Taster 12345 - Taster 3" Comment="" CmdOn="\xFD12345.BTN.19.STATUS.\v\xFE" CmdOff="" Unit="&lt;v.x&gt;" Analog="true" Text="false" Sensor="true" SourceValHigh="100" DestValHigh="100"/>
	<CommCmd Title="6-fach Taster 12345 - Taster 4" Comment="" CmdOn="\xFD12345.BTN.20.STATUS.\v\xFE" CmdOff="" Unit="&lt;v.x&gt;" Analog="true" Text="false" Sensor="true" SourceValHigh="100" DestValHigh="100"/>
	<CommCmd Title="6-fach Taster 12345 - Taster 5" Comment="" CmdOn="\xFD12345.BTN.21.STATUS.\v\xFE" CmdOff="" Unit="&lt;v.x&gt;" Analog="true" Text="false" Sensor="true" SourceValHigh="100" DestValHigh="100"/>
	<CommCmd Title="6-fach Taster 12345 - Taster 6" Comment="" CmdOn="\xFD12345.BTN.22.STATUS.\v\xFE" CmdOff="" Unit="&lt;v.x&gt;" Analog="true" Text="false" Sensor="true" SourceValHigh="100" DestValHigh="100"/>
	<CommCmd Title="6-fach Taster 12345 - Extern Taster 1" Comment="" CmdOn="\xFD12345.BTN.33.STATUS.\v\xFE" CmdOff="" Unit="&lt;v.x&gt;" Analog="true" Text="false" Sensor="true" SourceValHigh="100" DestValHigh="100"/>
	<CommCmd Title="6-fach Taster 12345 - Extern Taster 2" Comment="" CmdOn="\xFD12345.BTN.34.STATUS.\v\xFE" CmdOff="" Unit="&lt;v.x&gt;" Analog="true" Text="false" Sensor="true" SourceValHigh="100" DestValHigh="100"/>
	<CommCmd Title="6-fach Taster 12345 - Extern Taster 3" Comment="" CmdOn="\xFD12345.BTN.35.STATUS.\v\xFE" CmdOff="" Unit="&lt;v.x&gt;" Analog="true" Text="false" Sensor="true" SourceValHigh="100" DestValHigh="100"/>
	<CommCmd Title="6-fach Taster 12345 - Extern Taster 4" Comment="" CmdOn="\xFD12345.BTN.36.STATUS.\v\xFE" CmdOff="" Unit="&lt;v.x&gt;" Analog="true" Text="false" Sensor="true" SourceValHigh="100" DestValHigh="100"/>
	<CommCmd Title="6-fach Taster 12345 - Extern Taster 5" Comment="" CmdOn="\xFD12345.BTN.37.STATUS.\v\xFE" CmdOff="" Unit="&lt;v.x&gt;" Analog="true" Text="false" Sensor="true" SourceValHigh="100" DestValHigh="100"/>
	<CommCmd Title="6-fach Taster 12345 - Extern Taster 6" Comment="" CmdOn="\xFD12345.BTN.38.STATUS.\v\xFE" CmdOff="" Unit="&lt;v.x&gt;" Analog="true" Text="false" Sensor="true" SourceValHigh="100" DestValHigh="100"/>
	<CommCmd Title="6-fach Taster 12345 - Extern Led 1" Comment="" CmdOn="\xFD12345.LED.65.ON.&lt;v&gt;.0\xFE" CmdOff="\xFD12345.LED.65.OFF\xFE" Unit="" Analog="true" Text="false" Sensor="false" SourceValHigh="100" DestValHigh="100"/>
	<CommCmd Title="6-fach Taster 12345 - Extern Led 2" Comment="" CmdOn="\xFD12345.LED.66.ON.&lt;v&gt;.0\xFE" CmdOff="\xFD12345.LED.66.OFF\xFE" Unit="" Analog="true" Text="false" Sensor="false" SourceValHigh="100" DestValHigh="100"/>
	<CommCmd Title="6-fach Taster 12345 - Extern Led 3" Comment="" CmdOn="\xFD12345.LED.67.ON.&lt;v&gt;.0\xFE" CmdOff="\xFD12345.LED.67.OFF\xFE" Unit="" Analog="true" Text="false" Sensor="false" SourceValHigh="100" DestValHigh="100"/>
	<CommCmd Title="6-fach Taster 12345 - Extern Led 4" Comment="" CmdOn="\xFD12345.LED.68.ON.&lt;v&gt;.0\xFE" CmdOff="\xFD12345.LED.68.OFF\xFE" Unit="" Analog="true" Text="false" Sensor="false" SourceValHigh="100" DestValHigh="100"/>
	<CommCmd Title="6-fach Taster 12345 - Extern Led 5" Comment="" CmdOn="\xFD12345.LED.69.ON.&lt;v&gt;.0\xFE" CmdOff="\xFD12345.LED.69.OFF\xFE" Unit="" Analog="true" Text="false" Sensor="false" SourceValHigh="100" DestValHigh="100"/>
	<CommCmd Title="6-fach Taster 12345 - Extern Led 6" Comment="" CmdOn="\xFD12345.LED.70.ON.&lt;v&gt;.0\xFE" CmdOff="\xFD12345.LED.70.OFF\xFE" Unit="" Analog="true" Text="false" Sensor="false" SourceValHigh="100" DestValHigh="100"/>
	<CommCmd Title="6-fach Taster 12345 - RFID Leser" Comment="" CmdOn="\xFD12345.RFD.65.TAG_ID.\v\xFE" CmdOff="" Unit="&lt;v.x&gt;" Analog="false" Text="true" Sensor="true" SourceValHigh="100" DestValHigh="100"/>
	<CommCmd Title="6-fach Taster 12345 - RFID Leser" Comment="" CmdOn="\xFD12345.RFD.66.TAG_ID.\v\xFE" CmdOff="" Unit="&lt;v.x&gt;" Analog="false" Text="true" Sensor="true" SourceValHigh="100" DestValHigh="100"/>
	<CommCmd Title="6-fach Taster 12345 - RFID Leser" Comment="" CmdOn="\xFD12345.RFD.67.TAG_ID.\v\xFE" CmdOff="" Unit="&lt;v.x&gt;" Analog="false" Text="true" Sensor="true" SourceValHigh="100" DestValHigh="100"/>
	<CommCmd Title="6-fach Taster 12345 - RFID Leser" Comment="" CmdOn="\xFD12345.RFD.68.TAG_ID.\v\xFE" CmdOff="" Unit="&lt;v.x&gt;" Analog="false" Text="true" Sensor="true" SourceValHigh="100" DestValHigh="100"/>
	<CommCmd Title="6-fach Taster 12345 - RFID Leser" Comment="" CmdOn="\xFD12345.RFD.69.TAG_ID.\v\xFE" CmdOff="" Unit="&lt;v.x&gt;" Analog="false" Text="true" Sensor="true" SourceValHigh="100" DestValHigh="100"/>
	</Comm>
*)
END_ACTION

END_FUNCTION_BLOCK

// ---- POUs/RS485_Hausbus_FB/02_UniBaustein/fb_UniHBComOperator.TcPOU
(*======================================================================================================================================*)
(*//=============================================================================\\
||  _   _ _  __  _         _                        _   _                      ||
|| | \ | | |/ / / \  _   _| |_ ___  _ __ ___   __ _| |_(_) ___  _ __         ||
|| |  \| | ' / / _ \| | | | __/ _ \| '_ ` _ \ / _` | __| |/ _ \| '_ \        ||
|| | |\  | . \/ ___ \ |_| | || (_) | | | | | | (_| | |_| | (_) | | | |       ||
|| |_| \_|_|\_\_/  \_\__,_|\__\___/|_| |_| |_|\__,_|\__|_|\___/|_| |_|       ||
||                                                                             ||
\\=============================================================================//
fb_UniHBComOperator:		Soll ein neuer einfacher Universalbaustein für die Hausbus Kommunikation werden,
							er soll die Kommunikation innerhalb der Device Bausteine Standartisieren, sodass künftige änderungen
							einfach an allen Devices gleich erfolgen und nicht überall alles angepasst werden muss!	
						 *)
(*
Date          	| Version    	| created under        	| Author          	| Remark *)
(*====================================================================================================================================================*)
(*28/08/2025   	| 1.00      		| TC3		  		| N.Kersting       	| first release *)
(*28/08/2025   	| 1.01      		| TC3		  		| N.Kersting       	| Erster Test erfogreich *)
(*05/09/2025   	| 1.02      		| TC3		  		| N.Kersting       	| Implementierung eines Change Counters, Zählt Startups hoch/ Startup Afterreset ansteuerung geändert *)
(*13/09/2025   	| 1.03      		| TC3		  		| N.Kersting       	| Doku hinzugefügt *)
(*10/01/2026   	| 1.04      		| TC3		  		| N.Kersting       	| Check Ping Eingang hinzugefügt um das Ping prüfen auszuschalten *)
(*====================================================================================================================================================*)
FUNCTION_BLOCK fb_UniHBComOperator
VAR_INPUT
	I_stIdent			:ST_HausBus_Ident;		(* HausBus Ident Struktur *)
		
	I_bExtInputs		:BOOL := FALSE;			(* Benutzung der Externen Inputs Aktivieren *)
	I_bExecute			:BOOL;					(* Aktivierung der Operation des Geräts *)
	I_bPing				:BOOL;					(* Ping eingang *)
	I_bPingCheck		:BOOL := TRUE;			(* wenn aus, wird kein Ping verwendet *)
	I_bEventStartupDone	:BOOL;					(* Rückmeldung von den Eventbausteinen	*)
	I_bResetSendDone	:BOOL;					(* Rückmeldung vom Fifo, Reset befehl ausgeführt *)
	I_bStartupDone 		:BOOL;					(* Rückmeldung vom Device, Startup ausgeführt *)		
		
	I_tPingTimeout		:TIME := T#15S;			(* Zeit Parameter für Timeout Ping *)
	I_tStartupAfterReset :TIME := T#5S;			
	I_tReboot			:TIME := T#10S;			(* Verzögerungszeit nach dem Reset ausgeführt wurde *)	
	
END_VAR
VAR_OUTPUT
	Q_EState			:E_EnumHBDeviceOPMode;
	Q_bResetEvents		:BOOL;					(* Reset Events Startup *)
	Q_bExecuteEvents	:BOOL;					(* Events Startup Starten *)
	Q_bSendResetCmd		:BOOL;					(* Sende Reset zum Gerät *)
	Q_bStartupStart		:BOOL;					(* Startup Starten *)
	Q_bActivateSend		:BOOL;					(* Aktiviere Sendefunktion *)
	Q_bOP				:BOOL;					(* Gerät im OP Mode *)
	Q_bCom				:BOOL;					(* Verbindung zum Gerät aufgebaut *)
	Q_bError			:BOOL;					(* Gerät im Fehlerzustand *)
	Q_sState			:STRING;
	Q_dwChanges			:DWORD;
END_VAR
VAR
	(*================================================================*)
	(*	Funktionsbausteine *)
	(*================================================================*)
	fbPing				:fb_RS485PingCheck;
	r_trigStartupAfterReset	:r_trig;
	tonStartupAfterReset	:ton;
	tonResetDone			:ton;
	
	(*================================================================*)
	(*	Int Variablen *)
	(*================================================================*)
	i					:INT;
	dwChanges			:DWORD :=0;
	(*================================================================*)
	(*	String Variablen *)
	(*================================================================*)
	sDeviceStartup		:STRING;
	
	(*================================================================*)
	(*	Bool Variablen *)
	(*================================================================*)
	bResetEvents		:BOOL := FALSE;
	bExecuteEvents		:BOOL := FALSE;
	bSendResetCmd		:BOOL := FALSE;
	bStartupStart		:BOOL := FALSE;
	bStartUpCheckPing	:BOOL := FALSE;
	bPingOK				:BOOL := FALSE;
	bActivateSend		:BOOL := FALSE;
	bError				:BOOL := FALSE;
	(*================================================================*)
	(*	Enums  *)
	(*================================================================*)
	EnumHBDeviceOPMode	:E_EnumHBDeviceOPMode;
	
	
END_VAR

(*///////////////////////////////////////////////////////////*)
(* Startup Zurücksetzen Reset *)

(* Startup Automatisch Zurücksetzen bei Busverlust *)
tonStartupAfterReset(
	IN := NOT bPingOK
			AND bStartUpCheckPing
			AND NOT (EnumHBDeviceOPMode=E_HB_Device_WaitCom)
			AND NOT (EnumHBDeviceOPMode=E_HB_Device_Reset),	(* Neu, damit nicht immer wieder neugestartet wird -> Bootschleife verhindern*)
	PT:= I_tStartupAfterReset);

r_trigStartupAfterReset
	(CLK := tonStartupAfterReset.Q);
	
IF NOT I_bExecute
	OR r_trigStartupAfterReset.Q
THEN
	EnumHBDeviceOPMode := E_HB_Device_Init;
END_IF

tonResetDone(
	PT:= I_tReboot);
	
(*///////////////////////////////////////////////////////////*)
(* Reset Changes *)
IF NOT I_bExecute
	OR bResetChangesCounter_All
THEN
	dwChanges := 0;
END_IF

(*///////////////////////////////////////////////////////////*)
(*	Ping Dauerhaft Prüfen *)
fbPing(
	I_bPing:= 				I_bPing, 
	I_bExecute:= 			bStartUpCheckPing, 
	I_bAutoPing:= 			TRUE, 
	I_bAutoReset:= 			TRUE, 
	I_bReset:= 				NOT bStartUpCheckPing,  
	I_tPingTimeout:= 		I_tPingTimeout);

bPingOK := 	fbPing.Q_bComOk
			OR NOT I_bPingCheck;
(*///////////////////////////////////////////////////////////*)
(*	Device States *)
CASE EnumHBDeviceOPMode OF
(*///////////////////////////////////////////////////////////*)
E_HB_Device_Init:	

	sDeviceStartup := 'INIT';
	bResetEvents := TRUE;
	bExecuteEvents := FALSE;
	bSendResetCmd := FALSE;
	bStartupStart := FALSE;
	bStartUpCheckPing := FALSE;
	bActivateSend := FALSE;
	tonResetDone.IN := FALSE;
	
	IF I_bExecute
	THEN
		EnumHBDeviceOPMode := E_HB_Device_CheckID;
	END_IF

(*///////////////////////////////////////////////////////////*)	
E_HB_Device_CheckID:
	
	sDeviceStartup := 'Device ID Prüfen';
	
	IF I_stIdent.diID <> 0
	THEN
		IF NOT I_bEventStartupDone
		THEN
			EnumHBDeviceOPMode :=	E_HB_Device_EventStartup;
		END_IF
	ELSE
		sDeviceStartup := 'ERROR- Device ID Prüfen';
	END_IF
	
(*///////////////////////////////////////////////////////////*)	
E_HB_Device_EventStartup:
		
	sDeviceStartup := 'Startup Events';	
	bResetEvents := FALSE;
	bExecuteEvents := TRUE;	(* Muss immer an bleiben *)
	bStartUpCheckPing := TRUE;
	
	IF I_bEventStartupDone
	THEN
		sDeviceStartup := 'Startup Events- warte auf Reset False Flanke';	
		IF NOT I_bResetSendDone
		THEN
			EnumHBDeviceOPMode :=	E_HB_Device_Reset;
		END_IF
	END_IF
		
(*///////////////////////////////////////////////////////////*)	
E_HB_Device_Reset:
	
	sDeviceStartup := 'Reset Ausführen';	
	bActivateSend := TRUE;
	bSendResetCmd := TRUE;
	
	IF I_bResetSendDone
	THEN
		bSendResetCmd := FALSE;
		IF NOT I_bStartupDone
		THEN
			sDeviceStartup := 'Reset Ausgeführt- warte auf Startup False Flanke';
			EnumHBDeviceOPMode :=	E_HB_Device_WaitCom;
		END_IF
	END_IF
	
(*///////////////////////////////////////////////////////////*)	
E_HB_Device_WaitCom:

	sDeviceStartup := 'Warte auf Com';	
	tonResetDone.IN := TRUE;
	
	IF tonResetDone.Q
	THEN
		IF bPingOK
		THEN
			EnumHBDeviceOPMode :=	E_HB_Device_Startup;
		END_IF
	END_IF
	
(*///////////////////////////////////////////////////////////*)	
E_HB_Device_Startup:
	
	sDeviceStartup := 'Startup Ausführen';	
	bStartupStart := TRUE;
	
	IF I_bStartupDone
	THEN
		dwChanges := dwChanges +1;
		EnumHBDeviceOPMode :=	E_HB_Device_OP;
	END_IF
	
E_HB_Device_OP:
	sDeviceStartup := 'Gerät im OP Mode';	
	bStartupStart := FALSE;
END_CASE

(*///////////////////////////////////////////////////////////*)	
bError :=	(fbPing.Q_bTimeout 
			AND I_bPingCheck)
			AND I_stIdent.diID <> 0;
			
(*///////////////////////////////////////////////////////////*)	
(* Outputs *)
Q_EState 			:=	EnumHBDeviceOPMode;
Q_bResetEvents 		:=	bResetEvents;
Q_bExecuteEvents	:=	bExecuteEvents;
Q_bSendResetCmd		:=	bSendResetCmd;
Q_bStartupStart		:=	bStartupStart;
Q_bActivateSend		:=	bActivateSend;
Q_bCom				:=	bPingOK;
Q_bError			:=	bError;
Q_bOP				:=	(EnumHBDeviceOPMode =E_HB_Device_OP);
Q_sState			:=	sDeviceStartup;
Q_dwChanges			:=	dwChanges;

ACTION ac99_Doku:
(*=====================================================================*)
(*  Baustein: fb_UniHBComOperator                                      *)
(*  Zweck: Standardisiert den Lebenszyklus eines HausBus-Gerätes.      *)
(*  Fokus: Einheitliche Startup-/Reset-/Com- und Ping-Logik.           *)
(*---------------------------------------------------------------------*)
(*  Hauptablauf (Zustandsmaschine E_EnumHBDeviceOPMode):               *)
(*    1) E_HB_Device_Init         : Grundzustand, wartet auf Execute.  *)
(*    2) E_HB_Device_CheckID      : Prüft I_stIdent.diID <> 0.         *)
(*    3) E_HB_Device_EventStartup : Start-Events laufen (Events an).   *)
(*    4) E_HB_Device_Reset        : Reset-Kommando senden.             *)
(*    5) E_HB_Device_WaitCom      : Reboot-Zeit + Ping abwarten.       *)
(*    6) E_HB_Device_Startup      : Gerätestart (Device-spezifisch).   *)
(*    7) E_HB_Device_OP           : Gerät im Betriebsmodus.            *)
(*---------------------------------------------------------------------*)
(*  Übergänge (vereinfacht):                                           *)
(*    Init -> CheckID bei I_bExecute=TRUE                              *)
(*    CheckID -> EventStartup wenn ID gültig und Events nicht fertig   *)
(*    EventStartup -> Reset nach I_bEventStartupDone                   *)
(*    Reset -> WaitCom nach I_bResetSendDone                          *)
(*    WaitCom -> Startup nach Rebootzeit & Ping OK                     *)
(*    Startup -> OP bei I_bStartupDone                                 *)
(*    Kommunikationsverlust nach OP/Event/Startup -> Timeout -> Init   *)
(*---------------------------------------------------------------------*)
(*  Ping-/Com-Überwachung:                                             *)
(*    fb_RS485PingCheck läuft mit AutoPing + AutoReset.                *)
(*    bPingOK = Q_bCom; Timeout liefert Fehlerflag.                    *)
(*    tonStartupAfterReset triggert Rücksprung Init bei Pingverlust,   *)
(*    jedoch nicht während RESET / WAITCOM (verhindert Schleifen).     *)
(*---------------------------------------------------------------------*)
(*  Wichtige Eingänge:                                                 *)
(*    I_bExecute          : Gesamtablauf aktiv/inaktiv.                *)
(*    I_bPing             : Eingang für Ping-Auswertung.               *)
(*    I_bEventStartupDone : Events abgeschlossen.                      *)
(*    I_bResetSendDone    : Resetbefehl ausgeführt.                    *)
(*    I_bStartupDone      : Gerätestart fertig.                        *)
(*    Zeitparameter: I_tPingTimeout / I_tStartupAfterReset / I_tReboot *)
(*---------------------------------------------------------------------*)
(*  Wichtige Ausgänge:                                                 *)
(*    Q_EState        : Aktueller Enum-Zustand.                        *)
(*    Q_bResetEvents  : Events zurücksetzen (nur INIT).                *)
(*    Q_bExecuteEvents: Events aktiv halten (Startup-Phase).           *)
(*    Q_bSendResetCmd : Reset-Befehl senden (Puls in RESET).           *)
(*    Q_bStartupStart : Startsignal Gerätestart.                       *)
(*    Q_bActivateSend : Senden erlaubt (während RESET).                *)
(*    Q_bCom          : Kommunikation/Ping OK.                         *)
(*    Q_bOP           : Gerät im OP Mode.                              *)
(*    Q_bError        : Ping Timeout bei gültiger ID.                  *)
(*    Q_sState        : Textstatus für Diagnose.                       *)
(*    Q_dwChanges     : Zählt erfolgreiche Übergänge nach OP (Startup).*)
(*---------------------------------------------------------------------*)
(*  Change Counter:                                                    *)
(*    Erhöht bei Übergang Startup -> OP.                               *)
(*    Rücksetzung bei I_bExecute=FALSE.                                *)
(*---------------------------------------------------------------------*)
(*  Fehlerlogik:                                                       *)
(*    Q_bError = (Ping Timeout) AND (ID gültig).                       *)
(*    Ungültige ID nur im Text erkennbar (kein separates Flag).        *)
(*---------------------------------------------------------------------*)
(*  Robustheit:                                                        *)
(*    Schutz vor Reset-/Boot-Schleife durch Zustandseinschränkung      *)
(*    beim Auto-Restart (kein Trigger in RESET/WAITCOM).               *)
(*---------------------------------------------------------------------*)
(*  Erweiterungspotenzial (optional):                                  *)
(*    - Separater Fehlerzustand für ID=0.                              *)
(*    - Differenziertere Fehlercodes.                                  *)
(*    - Überlaufabsicherung Q_dwChanges.                               *)
(*    - Nutzung von I_bExtInputs (aktuell ungenutzt).                  *)
(*---------------------------------------------------------------------*)
(*  Einbindung (Kurz):                                                 *)
(*    1) Baustein mit Ident + Rückmeldeflags + Ping versorgen.         *)
(*    2) Auf Q_bSendResetCmd und Q_bStartupStart reagieren.            *)
(*    3) Betriebszustand über Q_EState / Q_bOP / Q_sState auswerten.   *)
(*---------------------------------------------------------------------*)
(*  Ziel: Einheitliche, wiederverwendbare Kommunikations- und          *)
(*  Startlogik für HausBus-Geräte mit minimalem Integrationsaufwand.  *)
(*=====================================================================*)
END_ACTION

END_FUNCTION_BLOCK

// ---- POUs/RS485_Hausbus_FB/02_UniBaustein/fb_RS485PingCheck.TcPOU
(*======================================================================================================================================*)
(*//=============================================================================\\
||  _   _ _  __  _         _                        _   _                      ||
|| | \ | | |/ / / \  _   _| |_ ___  _ __ ___   __ _| |_(_) ___  _ __         ||
|| |  \| | ' / / _ \| | | | __/ _ \| '_ ` _ \ / _` | __| |/ _ \| '_ \        ||
|| | |\  | . \/ ___ \ |_| | || (_) | | | | | | (_| | |_| | (_) | | | |       ||
|| |_| \_|_|\_\_/  \_\__,_|\__\___/|_| |_| |_|\__,_|\__|_|\___/|_| |_|       ||
||                                                                             ||
\\=============================================================================//
fb_RS485PingCheck:	Einfacher Universal Ping Baustein um von allerlei Geräten von haus-bus.de Kommunikation zu Checken über RS485 
				im gegensatz zum ComCheck Baustein wird hier nur gelesen, da es Geräte gibt, welche entweder Zyklich selbst 
				ein Lebenszeichen geben z.B. CYD oder die 6Fach Taster (Helligkeit, Temp, Luftfeuchtigkeit).
				Besonderheit bei dem 6Fach Taster ist: nach einem Reset werden immer auch StatusTelegramme gesendet. 
				Damit lässt sich dann auch festellen ob ein Taster Online ist. 
				Für die Aktoren ist dieser Baustein eher weniger geeignet, da es dort keine Zyklischen Telegramme gibt und 
				auch nach einem Reset keine Statustelegramme gesendet werden! 
				
				Der Baustein kann auch verwendet werden um einfach nur zu überwachen, ob ein Teilnehmer noch online ist über langen
				Zeitraum- Dafür muss der Timeout einfach sehr Hoch gestellt werden - z.B 120 Minuten und bAutoPing Aktiviert sein 
			
				Wenn I_bAutoPing nicht Aktiv ist, wird nur eine Ping überprüfung beim Aktivieren des Bausteins über I_bExecute 
				durchgeführt. Wenn die Prüfung erfolgreich ist, wird der Status Q_bComOk gesetzt. Der Status Q_bComOk wird erst durch 
				I_bReset wieder zurück gesetzt. 
				
				Wenn I_bAutoPing Aktiv ist, wird sobald der Baustein über I_bExecute gestartet wurde, und ein Ping Aufgebaut ist, 
				immer nach ablauf der Zeit: I_tPingTimeout erneut der Ping geprüft. Sollte der Ping nicht kommen, so wird nach ablauf der 
+				Zeit: I_tPingTimeout in den Timepout gesprungen. Dann kann nur über einen Reset durch: I_bReset erneut gestartet werden*)
(*
Date          	| Version    	| created under        	| Author          	| Remark *)
(*====================================================================================================================================================*)
(*28/08/2025   	| 1.00      		| TC3		  		| N.Kersting       | first release *)
(*04/09/2025   	| 1.01      		| TC3		  		| N.Kersting       | Etwas beschleunigter Ablauf wenn Ping in Step 999 kommt, wird erneut begonnen   *)
(*05/09/2025   	| 1.02      		| TC3		  		| N.Kersting       | Neuer Bugfix soll verhindern, dass bei Dynamischer Timeoutanpassung ein Verbindungsfehler auftritt   *)
(*====================================================================================================================================================*)
FUNCTION_BLOCK fb_RS485PingCheck
VAR_INPUT
	I_bPing				:BOOL;							(* Ping Event Empfangen *)
	I_bExecute			:BOOL;							(* Aktiviert den Ablauf *)
	I_bAutoPing			:BOOL;							(* Aktiviert die Automatische Prüfung, wenn aus- wird nur einmal beim Aktivieren über bExecute geprüft *)
	I_bAutoReset		:BOOL;							(* Aktiviert das Automatische wieder Quittieren wenn der Ping nicht empfangen wurde *)
	I_bReset			:BOOL;							(* Setzet den Ping und die Ablauf zurück *)
	I_tPingTimeout		:TIME := T#2S;					(* Zeit, bis der Ping gekommen sein muss *)
END_VAR
VAR_OUTPUT		
	Q_sState			:STRING;						(* Status  *)
	Q_bComOk			:BOOL;							(* Verbindung Aufgebaut *)
	Q_bTimeout			:BOOL;							(* Timeout  *)
END_VAR
VAR
	bResetCnt			:BOOL;
	tonTimeout			:ton;
	icntSymbole			:INT;
	iStep				:INT;
	i					:INT;
	bCOMMem				:BOOL;
	rTrigFailCount		:r_trig;
	dwCntFail			:DWORD;
	tPingTimeout		:TIME := T#15S;

END_VAR

(* Timeout Zeit *)
tonTimeout(
	PT:= tPingTimeout);

(* Ping Fehler Zählen *)	
rTrigFailCount();
	
(* Reset ausführen *)
IF I_bReset 
	OR NOT I_bExecute
THEN
	iStep := 0;	
END_IF

(* Timeout Counter auf 0 Setzen *)
IF bResetCnt
THEN
	dwCntFail := 0;
END_IF

(* Wenn timer aktiv und die Pingzeit ist Größer geworden, soll direkt die Zeitangepasst werden*)
IF 	I_tPingTimeout
	> tPingTimeout
	AND tonTimeout.IN
THEN
	tPingTimeout :=	I_tPingTimeout;
ELSIF
	I_tPingTimeout
	<> tPingTimeout
	AND NOT tonTimeout.IN
THEN
	tPingTimeout :=	I_tPingTimeout;
END_IF

(* Ablauf *)
CASE iStep OF
(*=========================================================*)	
0:	Q_sState := 'INIT';
	Q_bComOk := FALSE;
	bCOMMem := FALSE; (* Ping zurück setzen *)
	tonTimeout.IN := FALSE;
	Q_bTimeout := FALSE;
	rTrigFailCount.CLK := FALSE;
	
	IF I_bExecute
	THEN
		iStep := iStep +1;
	END_IF
	
(*=========================================================*)	
1:	Q_sState :=  'Warten auf Ping ';	
	tonTimeout.IN := TRUE;
	
	IF I_bPing
	THEN
		tonTimeout.IN := FALSE;
		bCOMMem := TRUE;
		iStep := 998;
	ELSIF
		tonTimeout.Q
	THEN
		tonTimeout.IN := FALSE;
		Q_bTimeout := TRUE;
		Q_bComOk := FALSE;
		Q_sState :=  'Timeout- Kein Ping empfangen';	
		iStep := -1;
	END_IF

(*=========================================================*)	
998: Q_sState :=  'Ping empfangen, Warte das String Leer ist';	
	tonTimeout.IN := TRUE;
	
	IF NOT I_bPing
	THEN
		tonTimeout.IN := FALSE;	(* Neu, hier zurücksetzen damit in 999 neu gestartet wird!*)
		iStep := 999;
	ELSIF
		tonTimeout.Q
	THEN
		tonTimeout.IN := FALSE;
		Q_bTimeout := TRUE;
		Q_bComOk := FALSE;
		Q_sState :=  'Timeout String wurde nicht geleert!';	
		iStep := -998;
	END_IF
	
(*=========================================================*)	
999: Q_sState :=  'Ping empfangen, erfolgreich Verbunden!';		
	Q_bComOk := TRUE;
	Q_bTimeout := FALSE;
	
	(* Die Verbindung wurde nun geprüft, kann aber nur über
		I_bReset wieder erneut geprüft werden ! *)
	
	IF I_bAutoPing
	THEN
		tonTimeout.IN := TRUE;
		
		IF tonTimeout.Q
			OR I_bPing	(* Neu- Soll den Ablauf etwas beschleunigen *)
		THEN
			tonTimeout.IN := FALSE;
				
			IF I_bExecute
			THEN
				iStep := 1;	(* Erneut Prüfen *)
			END_IF
		
		END_IF
	ELSE
		tonTimeout.IN := FALSE;
	END_IF
ELSE
(*=========================================================*)	
(*	Timeout *)	
	rTrigFailCount.CLK := TRUE;
	
	IF rTrigFailCount.Q
	THEN
		dwCntFail := dwCntFail+1;
	END_IF
	(*	Automatische Quittierung *)	
	IF 	I_bAutoReset
	THEN
		tonTimeout.IN := TRUE;
		
		IF tonTimeout.Q
			OR I_bPing
		THEN
			tonTimeout.IN := FALSE;
			
			IF I_bExecute
			THEN
				rTrigFailCount.CLK := FALSE;
				iStep := 1;	(* Erneut Prüfen *)
			END_IF
		END_IF
	END_IF
END_CASE

END_FUNCTION_BLOCK

// ---- POUs/RS485_Hausbus_FB/01_CYD/fb_BusTasterEvent.TcPOU
FUNCTION_BLOCK fb_BusTasterEvent
VAR_INPUT
	 I_sID         			:STRING(10);     // Geräte-ID (z.B. '12345')
	 I_sInstID				:STRING(2) 	:=	'17';
	 I_sReceivedString		:STRING(255);	
	 I_bFaultDetection		:BOOL := FALSE;		(* Soll erkennen, ob ein Telegramm für das zurücksetzen eines Tasters nicht gekommen ist *)
	 I_tFaultDetectTime		:TIME := T#10S;
END_VAR
VAR_OUTPUT
	Q_bOut					:BOOL;
END_VAR
VAR
	tonFaultInput			:ton;
	findString0				:STRING(255) ;
	findString1				:STRING(255) ;
END_VAR

(* Automatische Fehlererkennung *)

IF I_bFaultDetection
THEN
	tonFaultInput(
		IN := Q_bOut,
		PT := I_tFaultDetectTime);
END_IF

findString0 := CONCAT(I_sID,'.');
findString0 := CONCAT(findString0,'BTN');
findString0 := CONCAT(findString0,'.');
findString0 := CONCAT(findString0,I_sInstID);
findString0 := CONCAT(findString0,'.');
findString0 := CONCAT(findString0,'STATUS.0');

findString1 := CONCAT(I_sID,'.');
findString1 := CONCAT(findString1,'BTN');
findString1 := CONCAT(findString1,'.');
findString1 := CONCAT(findString1,I_sInstID);
findString1 := CONCAT(findString1,'.');
findString1 := CONCAT(findString1,'STATUS.1');

IF FIND(I_sReceivedString,findString0) >0 
	OR ( tonFaultInput.Q
		AND I_bFaultDetection)
THEN
	Q_bOut := FALSE;
ELSIF
	FIND(I_sReceivedString,findString1) >0 
THEN
	Q_bOut := TRUE;
END_IF

END_FUNCTION_BLOCK

// ---- POUs/RS485_Hausbus_FB/01_CYD/fb_CYDBus6F.TcPOU
(*======================================================================================================================================*)
(*FB_TasterBusSimple:	Einfache RS485 Kommunikation für Haus-bus.de Komponenten zum testen 	
						Achtung: Bei dem 6 Fach Taster ist zu Beachten, dass es nur 4 Externe EA/s gibt also 4 LEDs und 4 Taster *)
(*
Date          	| Version    	| created under        	| Author          	| Remark *)
(*====================================================================================================================================================*)
(*29/04/2025   	| 1.00      		| TC3		  		| N.Kersting       | first release *)
(*02/05/2025   	| 1.01      		| TC3		  		| N.Kersting       | Events für die Buttons werden erfolgreich verarbeitet *)
(*02/05/2025   	| 1.02      		| TC3		  		| N.Kersting       | Events für Temp, Helligkeit, Fuehctigkeit erfolgreich Implementier *)
(*02/05/2025   	| 1.03      		| TC3		  		| N.Kersting       | Set Schrittkette für Reset und LED Helligkeit erfolgreich Implementier*)
(*02/05/2025   	| 1.04      		| TC3		  		| N.Kersting       | In und Out Strukturen Implementiert und Startup nach Reset *)
(*02/05/2025   	| 1.05      		| TC3		  		| N.Kersting       | Pingabgfrage*)
(*02/05/2025   	| 1.06      		| TC3		  		| N.Kersting       | Reset Startup Implementiert*)
(*03/05/2025   	| 1.07      		| TC3		  		| N.Kersting       | Ping wird nun bei PLC Reset auch gestaret und Execute wird richtig verwendet*)
(*04/05/2025   	| 1.08      		| TC3		  		| N.Kersting       | Hintergrundbeleuchtung und Zähler für die Tatser Implementiert *)
(*04/05/2025   	| 1.09      		| TC3		  		| N.Kersting       | Neuen Baustein zum Einheitlichen versenden von Telegrammen Implementiert *)
(*05/05/2025   	| 2.00      		| TC3		  		| N.Kersting       | Komplett neuen Baustein, mit Externer Receive Auswertung und neuem Ping Baustein *)
(*06/05/2025   	| 2.01      		| TC3		  		| N.Kersting       | Externe LEDs Implementiert *)
(*07/05/2025   	| 2.02      		| TC3		  		| N.Kersting       | Im Startup wird nun auf die Device ID geachtet *)
(*08/05/2025   	| 2.03      		| TC3		  		| N.Kersting       | Externe LEDs sind nun Umschaltbar/ LEDs oder normaler Ausgang (Betriefft die Hintergrundbeleuchtung) -> Weniger Busauslastung *)
(*09/05/2025   	| 2.04      		| TC3		  		| N.Kersting       | Ping Versuche Implementiert mit Globalen Parametern *)
(*09/05/2025   	| 2.05      		| TC3		  		| N.Kersting       | Ping für Taster nun Auch automatisch durch Empfang von sämtlichen Telegrammen*)
(*09/05/2025   	| 2.06      		| TC3		  		| N.Kersting       | Bugfix im Startup Angepasst! nur noch Hintergrundbeleuchtung setzen! *)
(*10/05/2025   	| 3.00      		| TC3		  		| N.Kersting       | Umstellung auf Externe FiFo Sendebaustein *)
(*13/05/2025   	| 3.01      		| TC3		  		| N.Kersting       | Viele Bugs gefixt, bei Änderung der Ausgängen wird nun eine Anforderung gesetzt  *)
(*13/05/2025   	| 3.02      		| TC3		  		| N.Kersting       | Test für Github *)
(*22/05/2025   	| 3.03      		| TC3		  		| N.Kersting       | Grundaufbau vom BusTaster, jetzt allerdings für ein CYD mit den gleichen Funktionen *)
(*22/05/2025   	| 3.04      		| TC3		  		| N.Kersting       | ServiceFunktionen für CYD Hinzugefügt (Wifi und Webserver Starten)*)
(*23/05/2025   	| 3.05      		| TC3		  		| N.Kersting       | Neue eigene Input Struktur für das CYD Implementiert*)
(*23/05/2025   	| 3.06      		| TC3		  		| N.Kersting       | Auto - Input Fault Detection implementiert (Wenn Taster zu lange aktiviert bleibt ) *)
(*26/05/2025   	| 3.07      		| TC3		  		| N.Kersting       | Updaten im Com Check Baustein, der Zyklische Ping vom CYD wird nun erkannt ) *)
(*28/05/2025   	| 3.08      		| TC3		  		| N.Kersting       | Neuen Einfachen Ping Baustein, welcher nicht sendet, nur auswertet implementiert *)
(*09/09/2025   	| 3.09      		| TC3		  		| N.Kersting       | ---Alles wichtige Deaktiviert --- Warten auf neues Releas CYD *)
(*====================================================================================================================================================*)
FUNCTION_BLOCK fb_CYDBus6F
VAR_INPUT
	I_tReceiveTimeout	:TIME;
	I_iMaxPingTry		:INT;
	I_bUsePing			:BOOL;
	I_tPingTime			:TIME := T#15S;
	I_bFiFoDone			:BOOL;
	I_FifoID			:INT;
	I_bPingStart		:BOOL;						(* Ping Done vom Vorheriegen*)
	I_stInput			:ST_BusCYD6F_Input;
	I_StringReceived	:STRING(255);
END_VAR
VAR_OUTPUT
	Q_sFiFoSend			:STRING(255);
   	Q_stOutput			:ST_BusTaster6F_Output;
	Q_stCnt				:ST_BusTaster6F_Cnt;
END_VAR
VAR
(*----------------------------------------------*)
(* Interne Parameter*)
(*----------------------------------------------*)		
	bSetExecute			:BOOL := TRUE;				(* Aktiviert die Schrittketten, welche Telegramme versenden *)
	bCheckPing			:BOOL := TRUE;				(* Ping Checken Schrittkette Aktivieren *)
	sStartZeichen		:BYTE := 16#FD;				(* Startzeichen Präfix *)
	sEndZeichen			:BYTE := 16#FE;				(* Endzeichen Suffix *)
	iAnzResetSend		:INT := 2;					(* Anzahl der Sendeversuche bei Reset *)
	tPingTimer			:TIME:= T#5S;				(* Zeit, bis wiederholend der Ping versendet wird *)
	tReceiveTimeout		:TIME:= T#2S;				(* Zeit, bis die Event Schrittkette für das Empfangen Automatisch neu Startet*)
	tStartupLEDOn		:TIME:= T#4S;				(* Zeit, wie Lange die LEDS beim Startup kurz eingeschaltet werden *)
	tResetTimeout		:TIME:= T#25S;				(* Zeit, bis bei einem Reset es zu einem Fehler kommt, wenn kein Ping empfangen wird *)
	tResetReboot		:TIME:= T#10S;				(* Zeit, die nach einem Reset Abgewaretet wird damit das Gerät neustarten kann*)
	tResetStartup		:TIME:= T#5S;				(* Zeit, die nach einem Reset Abgewaretet wird bis ein Startup ausgeführt wird nach dem erhalt des Pings vom Gerät*)
	tStartupAfterReset	:TIME := T#5S;				(* Zeit, wann das Startup Zurückgesetzt wird, wenn der Ping verloren wird *)
	bInputFaultDetect	:BOOL := TRUE;				(* Prüft die Eingänge ob sie zu lange geschaltet wurden und führt ein reset des eingangs aus *)
	tInputFaultDetect	:TIME := T#10S;				(* Prüft die Eingänge ob sie zu lange geschaltet wurden und führt ein reset des eingangs aus *)
(*----------------------------------------------*)
(*	Service Funktionen Aktivieren *)
(*----------------------------------------------*)	
	bWebServer			:BOOL := FALSE;				(* zuerst funktion auswählen (bWebserver/ bWifi, bService) und dann mit bStartServiceMode ausführen *)
	bWifi				:BOOL := FALSE;				(* zuerst funktion auswählen (bWebserver/ bWifi, bService) und dann mit bStartServiceMode ausführen *)
	bService			:BOOL := FALSE;				(* zuerst funktion auswählen (bWebserver/ bWifi, bService) und dann mit bStartServiceMode ausführen *)
	(*	*)
	bStartServiceMode	:BOOL := FALSE;				(* zuerst ServiceMode Aktivieren und dann mit bStartServiceMode ausführen *)
	
	(* Speichern der zustände *)
	bMemWebServer		:BOOL;
	bMemWifi			:BOOL;
	bMemService			:BOOL;
	
